C05467=1038.673,-19.331,418.240,169.034,37.910,157.122
C05468=1038.665,-19.613,418.256,169.031,37.909,157.122
C05469=1038.659,-19.895,418.271,169.029,37.909,157.121
C05470=1038.651,-20.177,418.287,169.026,37.909,157.121
C05471=1038.645,-20.426,418.300,169.024,37.909,157.121
C05472=1038.639,-20.676,418.314,169.022,37.908,157.121
C05473=1038.632,-20.925,418.328,169.019,37.908,157.121
C05474=1038.625,-21.175,418.342,169.017,37.908,157.121
C05475=1038.620,-21.425,418.356,169.014,37.907,157.121
C05476=1038.613,-21.674,418.370,169.012,37.907,157.121
C05477=1038.607,-21.923,418.384,169.010,37.907,157.121
C05478=1038.600,-22.173,418.398,169.008,37.907,157.121
C05479=1038.594,-22.423,418.411,169.006,37.906,157.121
C05480=1038.588,-22.672,418.426,169.004,37.906,157.121
C05481=1038.582,-22.922,418.439,169.001,37.906,157.120
C05482=1038.575,-23.171,418.453,168.999,37.905,157.120
C05483=1038.569,-23.421,418.467,168.997,37.905,157.120
C05484=1038.563,-23.670,418.480,168.995,37.905,157.120
C05485=1038.556,-23.920,418.494,168.993,37.905,157.120
C05486=1038.551,-24.169,418.508,168.990,37.904,157.120
C05487=1038.544,-24.419,418.522,168.988,37.904,157.120
C05488=1038.538,-24.669,418.535,168.986,37.904,157.120
C05489=1038.532,-24.918,418.549,168.984,37.904,157.120
C05490=1038.525,-25.167,418.563,168.981,37.903,157.120
C05491=1038.519,-25.417,418.577,168.978,37.903,157.120
C05492=1038.513,-25.666,418.591,168.976,37.903,157.119
C05493=1038.506,-25.916,418.604,168.974,37.902,157.119
C05494=1038.500,-26.166,418.617,168.972,37.902,157.119
C05495=1038.494,-26.416,418.632,168.970,37.902,157.119
C05496=1038.488,-26.665,418.645,168.967,37.902,157.119
C05497=1038.482,-26.915,418.659,168.965,37.901,157.119
C05498=1038.476,-27.165,418.672,168.963,37.901,157.119
C05499=1038.469,-27.414,418.686,168.961,37.901,157.119
C05500=1038.463,-27.664,418.699,168.958,37.901,157.119
C05501=1038.456,-27.913,418.713,168.956,37.900,157.119
C05502=1038.450,-28.162,418.727,168.954,37.900,157.119
C05503=1038.443,-28.412,418.740,168.952,37.900,157.119
C05504=1038.437,-28.661,418.753,168.949,37.900,157.119
C05505=1038.431,-28.911,418.766,168.947,37.900,157.119
C05506=1038.425,-29.161,418.780,168.944,37.899,157.118
C05507=1038.419,-29.410,418.794,168.942,37.899,157.118
C05508=1038.412,-29.660,418.807,168.939,37.900,157.118
C05509=1038.406,-29.910,418.820,168.937,37.899,157.118
C05510=1038.399,-30.159,418.834,168.935,37.899,157.118
C05511=1038.393,-30.409,418.847,168.933,37.899,157.118
C05512=1038.386,-30.658,418.861,168.930,37.899,157.118
C05513=1038.380,-30.907,418.874,168.928,37.899,157.118
C05514=1038.373,-31.157,418.888,168.926,37.898,157.118
C05515=1038.367,-31.407,418.901,168.924,37.898,157.118
C05516=1038.361,-31.656,418.914,168.921,37.898,157.118
C05517=1038.355,-31.905,418.927,168.919,37.898,157.118
C05518=1038.348,-32.155,418.941,168.917,37.898,157.118
C05519=1038.343,-32.405,418.954,168.915,37.897,157.118
C05520=1038.336,-32.655,418.967,168.912,37.897,157.117
C05521=1038.330,-32.905,418.981,168.910,37.897,157.117
C05522=1038.323,-33.154,418.994,168.908,37.897,157.117
C05523=1038.317,-33.403,419.008,168.906,37.897,157.117
C05524=1038.311,-33.652,419.021,168.903,37.896,157.117
C05525=1038.304,-33.902,419.034,168.901,37.896,157.117
C05526=1038.298,-34.152,419.047,168.899,37.896,157.117
C05527=1038.292,-34.401,419.060,168.895,37.896,157.117
C05528=1038.286,-34.651,419.074,168.893,37.896,157.117
C05529=1038.279,-34.901,419.087,168.891,37.895,157.117
C05530=1038.273,-35.150,419.100,168.889,37.896,157.117
C05531=1038.266,-35.432,419.115,168.886,37.896,157.117
C05532=1038.259,-35.712,419.130,168.883,37.895,157.117
C05533=1038.252,-35.993,419.145,168.881,37.895,157.117
C05534=1038.245,-36.275,419.160,168.878,37.895,157.116
C05535=1038.239,-36.524,419.173,168.876,37.895,157.116
C05536=1038.233,-36.773,419.186,168.874,37.895,157.116
C05537=1038.227,-37.023,419.199,168.872,37.894,157.116
C05538=1038.220,-37.273,419.212,168.869,37.894,157.116
C05539=1038.214,-37.523,419.226,168.867,37.894,157.116
C05540=1038.208,-37.772,419.239,168.865,37.894,157.116
C05541=1038.202,-38.022,419.252,168.862,37.894,157.116
C05542=1038.195,-38.271,419.265,168.860,37.893,157.116
C05543=1038.189,-38.520,419.278,168.858,37.893,157.116
C05544=1038.183,-38.771,419.291,168.856,37.893,157.116
C05545=1038.177,-39.020,419.304,168.853,37.893,157.116
C05546=1038.170,-39.269,419.318,168.851,37.893,157.116
C05547=1038.164,-39.519,419.330,168.849,37.893,157.116
C05548=1038.157,-39.768,419.343,168.846,37.893,157.116
C05549=1038.151,-40.019,419.356,168.843,37.893,157.116
C05550=1038.145,-40.268,419.369,168.841,37.893,157.116
C05551=1038.139,-40.518,419.382,168.838,37.893,157.116
C05552=1038.132,-40.767,419.394,168.836,37.893,157.116
C05553=1038.126,-41.016,419.407,168.834,37.893,157.116
C05554=1038.120,-41.266,419.420,168.831,37.892,157.115
C05555=1038.113,-41.516,419.434,168.829,37.892,157.115
C05556=1038.106,-41.766,419.446,168.827,37.893,157.115
C05557=1038.100,-42.015,419.459,168.824,37.893,157.115
C05558=1038.094,-42.265,419.471,168.822,37.892,157.115
C05559=1038.088,-42.514,419.485,168.820,37.892,157.115
C05560=1038.082,-42.764,419.497,168.817,37.892,157.115
C05561=1038.075,-43.013,419.510,168.815,37.892,157.115
C05562=1038.069,-43.263,419.522,168.813,37.892,157.115
C05563=1038.062,-43.513,419.536,168.810,37.892,157.115
C05564=1038.056,-43.763,419.549,168.808,37.892,157.115
C05565=1038.050,-44.012,419.561,168.805,37.892,157.115
C05566=1038.044,-44.261,419.574,168.803,37.892,157.115
C05567=1038.038,-44.511,419.586,168.801,37.892,157.115
C05568=1038.031,-44.761,419.600,168.798,37.892,157.115
C05569=1038.025,-45.010,419.612,168.796,37.892,157.115
C05570=1038.019,-45.259,419.625,168.794,37.892,157.115
C05571=1038.013,-45.509,419.638,168.791,37.892,157.115
C05572=1038.007,-45.759,419.650,168.789,37.891,157.115
C05573=1038.000,-46.008,419.663,168.787,37.891,157.114
C05574=1037.994,-46.258,419.675,168.784,37.891,157.114
C05575=1037.988,-46.508,419.688,168.782,37.892,157.114
C05576=1037.982,-46.757,419.701,168.780,37.892,157.114
C05577=1037.975,-47.007,419.713,168.777,37.891,157.114
C05578=1037.969,-47.256,419.726,168.775,37.891,157.114
C05579=1037.963,-47.506,419.739,168.773,37.891,157.114
C05580=1037.956,-47.755,419.751,168.770,37.891,157.114
C05581=1037.950,-48.005,419.764,168.768,37.891,157.114
C05582=1037.944,-48.255,419.777,168.764,37.891,157.114
C05583=1037.938,-48.504,419.789,168.762,37.891,157.114
C05584=1037.932,-48.754,419.801,168.760,37.891,157.114
C05585=1037.926,-49.003,419.814,168.757,37.891,157.114
C05586=1037.920,-49.253,419.827,168.755,37.891,157.114
C05587=1037.914,-49.503,419.840,168.753,37.891,157.114
C05588=1037.907,-49.752,419.852,168.750,37.891,157.114
C05589=1037.901,-50.002,419.865,168.748,37.891,157.114
C05590=1037.895,-50.252,419.877,168.746,37.891,157.114
C05591=1037.888,-50.501,419.889,168.743,37.891,157.114
C05592=1037.882,-50.751,419.902,168.741,37.891,157.114
C05593=1037.875,-51.000,419.915,168.738,37.891,157.114
C05594=1037.870,-51.250,419.927,168.736,37.891,157.114
C05595=1037.862,-51.532,419.940,168.733,37.891,157.114
C05596=1037.854,-51.813,419.955,168.730,37.891,157.114
C05597=1037.847,-52.095,419.968,168.728,37.892,157.114
C05598=1037.841,-52.376,419.982,168.725,37.892,157.114
C05599=1037.834,-52.626,419.994,168.722,37.892,157.114
C05600=1037.827,-52.875,420.006,168.720,37.892,157.114
C05601=1037.821,-53.125,420.019,168.718,37.892,157.114
C05602=1037.815,-53.375,420.031,168.715,37.892,157.113
C05603=1037.809,-53.624,420.043,168.713,37.892,157.113
C05604=1037.802,-53.874,420.055,168.710,37.892,157.113
C05605=1037.796,-54.124,420.067,168.708,37.892,157.113
C05606=1037.790,-54.373,420.080,168.705,37.892,157.113
C05607=1037.783,-54.623,420.092,168.703,37.893,157.114
C05608=1037.776,-54.873,420.104,168.701,37.893,157.113
C05609=1037.770,-55.122,420.116,168.698,37.893,157.113
C05610=1037.764,-55.372,420.128,168.696,37.893,157.113
C05611=1037.757,-55.622,420.140,168.693,37.893,157.113
C05612=1037.751,-55.872,420.153,168.691,37.894,157.113
C05613=1037.745,-56.121,420.165,168.688,37.894,157.113
C05614=1037.739,-56.370,420.176,168.686,37.894,157.113
C05615=1037.733,-56.620,420.189,168.683,37.894,157.113
C05616=1037.726,-56.869,420.201,168.681,37.894,157.113
C05617=1037.719,-57.119,420.213,168.679,37.894,157.113
C05618=1037.713,-57.369,420.225,168.676,37.894,157.113
C05619=1037.707,-57.618,420.237,168.674,37.894,157.113
C05620=1037.700,-57.868,420.249,168.671,37.894,157.113
C05621=1037.694,-58.118,420.262,168.669,37.895,157.113
C05622=1037.688,-58.367,420.273,168.666,37.895,157.113
C05623=1037.682,-58.617,420.285,168.664,37.895,157.113
C05624=1037.676,-58.867,420.297,168.661,37.895,157.113
C05625=1037.669,-59.116,420.309,168.659,37.895,157.113
C05626=1037.663,-59.366,420.321,168.656,37.895,157.113
C05627=1037.657,-59.616,420.334,168.654,37.896,157.113
C05628=1037.651,-59.865,420.345,168.652,37.896,157.113
C05629=1037.644,-60.114,420.357,168.649,37.896,157.113
C05630=1037.638,-60.365,420.369,168.647,37.896,157.113
C05631=1037.632,-60.614,420.381,168.644,37.896,157.113
C05632=1037.625,-60.864,420.393,168.642,37.897,157.113
C05633=1037.619,-61.113,420.405,168.639,37.897,157.113
C05634=1037.613,-61.363,420.417,168.637,37.897,157.113
C05635=1037.607,-61.613,420.428,168.634,37.897,157.113
C05636=1037.600,-61.862,420.440,168.632,37.897,157.113
C05637=1037.595,-62.112,420.453,168.629,37.897,157.113
C05638=1037.588,-62.361,420.465,168.627,37.897,157.113
C05639=1037.582,-62.611,420.476,168.624,37.897,157.113
C05640=1037.575,-62.861,420.488,168.622,37.897,157.113
C05641=1037.569,-63.111,420.500,168.619,37.897,157.113
C05642=1037.563,-63.360,420.512,168.617,37.898,157.113
C05643=1037.557,-63.609,420.524,168.614,37.898,157.113
C05644=1037.551,-63.860,420.536,168.612,37.898,157.113
C05645=1037.545,-64.109,420.547,168.610,37.898,157.113
C05646=1037.538,-64.358,420.559,168.607,37.899,157.113
C05647=1037.532,-64.608,420.570,168.605,37.899,157.113
C05648=1037.526,-64.858,420.583,168.602,37.899,157.113
C05649=1037.520,-65.107,420.595,168.600,37.899,157.113
C05650=1037.514,-65.357,420.606,168.597,37.899,157.113
C05651=1037.507,-65.607,420.618,168.595,37.900,157.113
C05652=1037.502,-65.856,420.630,168.592,37.900,157.113
C05653=1037.495,-66.106,420.641,168.590,37.900,157.113
C05654=1037.489,-66.356,420.653,168.587,37.900,157.113
C05655=1037.483,-66.605,420.665,168.585,37.900,157.113
C05656=1037.477,-66.855,420.677,168.582,37.900,157.113
C05657=1037.470,-67.105,420.689,168.580,37.900,157.113
C05658=1037.465,-67.354,420.699,168.577,37.900,157.113
C05659=1037.457,-67.637,420.714,168.574,37.901,157.113
C05660=1037.450,-67.920,420.727,168.572,37.901,157.113
C05661=1037.444,-68.202,420.740,168.569,37.901,157.113
C05662=1037.437,-68.485,420.753,168.566,37.901,157.113
C05663=1037.431,-68.735,420.765,168.564,37.901,157.113
C05664=1037.425,-68.985,420.776,168.561,37.902,157.113
C05665=1037.419,-69.234,420.788,168.559,37.902,157.113
C05666=1037.412,-69.484,420.799,168.556,37.902,157.113
C05667=1037.406,-69.733,420.811,168.554,37.902,157.113
C05668=1037.401,-69.984,420.823,168.551,37.903,157.113
C05669=1037.394,-70.233,420.835,168.549,37.903,157.113
C05670=1037.388,-70.483,420.845,168.546,37.903,157.113
C05671=1037.382,-70.732,420.857,168.544,37.903,157.113
C05672=1037.377,-70.982,420.869,168.541,37.903,157.113
C05673=1037.370,-71.232,420.881,168.539,37.904,157.113
C05674=1037.364,-71.481,420.892,168.536,37.904,157.113
C05675=1037.358,-71.731,420.904,168.534,37.904,157.113
C05676=1037.351,-71.981,420.915,168.531,37.904,157.113
C05677=1037.346,-72.231,420.926,168.529,37.904,157.113
C05678=1037.340,-72.480,420.938,168.526,37.904,157.113
C05679=1037.334,-72.730,420.949,168.524,37.905,157.113
C05680=1037.327,-72.979,420.961,168.521,37.905,157.113
C05681=1037.321,-73.229,420.972,168.519,37.905,157.113
C05682=1037.315,-73.479,420.985,168.516,37.905,157.113
C05683=1037.310,-73.728,420.996,168.514,37.905,157.113
C05684=1037.303,-73.978,421.007,168.511,37.905,157.113
C05685=1037.297,-74.227,421.018,168.508,37.906,157.113
C05686=1037.291,-74.477,421.030,168.506,37.906,157.113
C05687=1037.285,-74.727,421.040,168.503,37.906,157.113
C05688=1037.279,-74.977,421.052,168.501,37.907,157.113
C05689=1037.273,-75.226,421.063,168.498,37.907,157.113
C05690=1037.267,-75.476,421.075,168.496,37.908,157.113
C05691=1037.261,-75.726,421.085,168.493,37.908,157.113
C05692=1037.254,-75.975,421.097,168.491,37.908,157.113
C05693=1037.248,-76.225,421.108,168.488,37.909,157.113
C05694=1037.242,-76.475,421.120,168.485,37.909,157.113
C05695=1037.236,-76.724,421.130,168.483,37.909,157.113
C05696=1037.229,-76.974,421.142,168.480,37.910,157.113
C05697=1037.223,-77.223,421.153,168.478,37.910,157.113
C05698=1037.217,-77.473,421.164,168.475,37.911,157.113
C05699=1037.211,-77.723,421.175,168.473,37.911,157.113
C05700=1037.205,-77.973,421.186,168.470,37.911,157.113
C05701=1037.199,-78.222,421.198,168.468,37.911,157.113
C05702=1037.192,-78.472,421.209,168.465,37.912,157.113
C05703=1037.187,-78.722,421.220,168.462,37.912,157.113
C05704=1037.180,-78.972,421.231,168.460,37.912,157.113
C05705=1037.175,-79.221,421.242,168.457,37.913,157.113
C05706=1037.169,-79.471,421.253,168.455,37.913,157.113
C05707=1037.162,-79.721,421.263,168.452,37.913,157.113
C05708=1037.156,-79.970,421.274,168.450,37.913,157.113
C05709=1037.149,-80.220,421.286,168.448,37.914,157.113
C05710=1037.144,-80.469,421.297,168.445,37.915,157.113
C05711=1037.137,-80.719,421.308,168.443,37.915,157.113
C05712=1037.131,-80.969,421.319,168.440,37.916,157.113
C05713=1037.125,-81.219,421.330,168.437,37.916,157.113
C05714=1037.118,-81.468,421.340,168.435,37.917,157.113
C05715=1037.112,-81.718,421.351,168.432,37.917,157.113
C05716=1037.106,-81.968,421.362,168.430,37.918,157.114
C05717=1037.099,-82.217,421.373,168.427,37.918,157.114
C05718=1037.093,-82.467,421.384,168.424,37.918,157.114
C05719=1037.087,-82.716,421.395,168.422,37.919,157.114
C05720=1037.080,-82.966,421.405,168.419,37.919,157.114
C05721=1037.075,-83.216,421.416,168.417,37.920,157.114
C05722=1037.069,-83.465,421.427,168.414,37.920,157.114
C05723=1037.062,-83.751,421.439,168.411,37.921,157.114
C05724=1037.054,-84.036,421.452,168.408,37.922,157.114
C05725=1037.047,-84.321,421.464,168.405,37.922,157.114
C05726=1037.040,-84.606,421.476,168.402,37.922,157.114
C05727=1037.034,-84.855,421.486,168.399,37.923,157.114
C05728=1037.028,-85.105,421.497,168.397,37.923,157.114
C05729=1037.022,-85.355,421.508,168.394,37.924,157.114
C05730=1037.015,-85.604,421.519,168.391,37.925,157.114
C05731=1037.009,-85.854,421.529,168.389,37.925,157.114
C05732=1037.003,-86.104,421.541,168.387,37.926,157.114
C05733=1036.997,-86.354,421.550,168.385,37.926,157.114
C05734=1036.991,-86.603,421.561,168.382,37.927,157.114
C05735=1036.985,-86.853,421.572,168.379,37.927,157.114
C05736=1036.978,-87.102,421.583,168.377,37.927,157.114
C05737=1036.973,-87.352,421.594,168.374,37.928,157.114
C05738=1036.965,-87.602,421.604,168.371,37.928,157.114
C05739=1036.960,-87.852,421.614,168.369,37.929,157.115
C05740=1036.954,-88.101,421.625,168.366,37.930,157.115
C05741=1036.948,-88.351,421.636,168.364,37.930,157.115
C05742=1036.941,-88.601,421.647,168.361,37.931,157.115
C05743=1036.935,-88.850,421.657,168.358,37.931,157.115
C05744=1036.930,-89.100,421.667,168.356,37.931,157.115
C05745=1036.924,-89.350,421.678,168.353,37.932,157.115
C05746=1036.917,-89.599,421.689,168.350,37.933,157.115
C05747=1036.911,-89.849,421.700,168.348,37.933,157.115
C05748=1036.905,-90.099,421.709,168.345,37.934,157.115
C05749=1036.899,-90.348,421.720,168.342,37.934,157.115
C05750=1036.893,-90.598,421.731,168.340,37.935,157.115
C05751=1036.887,-90.848,421.741,168.337,37.935,157.115
C05752=1036.881,-91.098,421.752,168.335,37.936,157.115
C05753=1036.874,-91.347,421.762,168.332,37.936,157.115
C05754=1036.869,-91.596,421.773,168.330,37.937,157.115
C05755=1036.863,-91.847,421.783,168.328,37.937,157.115
C05756=1036.856,-92.096,421.794,168.325,37.938,157.115
C05757=1036.850,-92.346,421.805,168.322,37.939,157.115
C05758=1036.844,-92.596,421.814,168.320,37.939,157.115
C05759=1036.838,-92.845,421.825,168.317,37.940,157.116
C05760=1036.832,-93.096,421.835,168.314,37.940,157.116
C05761=1036.826,-93.345,421.846,168.312,37.940,157.116
C05762=1036.820,-93.595,421.857,168.309,37.941,157.116
C05763=1036.814,-93.844,421.866,168.306,37.942,157.116
C05764=1036.808,-94.094,421.877,168.304,37.942,157.116
C05765=1036.802,-94.344,421.887,168.301,37.943,157.116
C05766=1036.796,-94.593,421.898,168.298,37.944,157.116
C05767=1036.789,-94.843,421.908,168.296,37.944,157.116
C05768=1036.784,-95.093,421.918,168.293,37.944,157.116
C05769=1036.778,-95.343,421.929,168.291,37.945,157.116
C05770=1036.772,-95.592,421.939,168.288,37.946,157.116
C05771=1036.766,-95.842,421.950,168.285,37.946,157.116
C05772=1036.760,-96.092,421.959,168.283,37.947,157.116
C05773=1036.754,-96.341,421.970,168.281,37.948,157.116
C05774=1036.748,-96.591,421.980,168.277,37.948,157.116
C05775=1036.742,-96.841,421.991,168.276,37.948,157.116
C05776=1036.736,-97.091,422.001,168.273,37.949,157.116
C05777=1036.730,-97.341,422.011,168.270,37.949,157.116
C05778=1036.724,-97.590,422.021,168.268,37.950,157.117
C05779=1036.718,-97.840,422.032,168.265,37.951,157.117
C05780=1036.712,-98.090,422.041,168.262,37.952,157.117
C05781=1036.706,-98.339,422.051,168.260,37.952,157.117
C05782=1036.700,-98.589,422.062,168.257,37.953,157.117
C05783=1036.694,-98.839,422.071,168.254,37.954,157.117
C05784=1036.687,-99.088,422.082,168.251,37.955,157.117
C05785=1036.682,-99.338,422.092,168.249,37.955,157.117
C05786=1036.676,-99.588,422.101,168.246,37.955,157.117
C05787=1036.668,-99.874,422.113,168.243,37.956,157.117
C05788=1036.661,-100.162,422.125,168.240,37.957,157.117
C05789=1036.654,-100.449,422.136,168.238,37.958,157.117
C05790=1036.647,-100.737,422.148,168.235,37.959,157.118
C05791=1036.641,-100.987,422.158,168.232,37.959,157.118
C05792=1036.635,-101.236,422.168,168.229,37.960,157.118
C05793=1036.629,-101.486,422.178,168.226,37.961,157.118
C05794=1036.623,-101.736,422.187,168.224,37.962,157.118
C05795=1036.617,-101.986,422.197,168.221,37.962,157.118
C05796=1036.611,-102.235,422.208,168.218,37.963,157.118
C05797=1036.605,-102.485,422.217,168.216,37.964,157.118
C05798=1036.598,-102.734,422.227,168.213,37.965,157.118
C05799=1036.593,-102.984,422.238,168.210,37.965,157.118
C05800=1036.586,-103.234,422.247,168.208,37.966,157.118
C05801=1036.580,-103.484,422.257,168.205,37.967,157.118
C05802=1036.575,-103.734,422.267,168.203,37.968,157.119
C05803=1036.569,-103.983,422.277,168.200,37.969,157.119
C05804=1036.562,-104.233,422.287,168.198,37.969,157.119
C05805=1036.556,-104.482,422.296,168.195,37.970,157.119
C05806=1036.550,-104.732,422.306,168.192,37.971,157.119
C05807=1036.544,-104.982,422.316,168.190,37.972,157.119
C05808=1036.538,-105.232,422.326,168.187,37.972,157.119
C05809=1036.532,-105.482,422.335,168.184,37.972,157.119
C05810=1036.526,-105.731,422.346,168.181,37.973,157.119
C05811=1036.521,-105.981,422.355,168.179,37.974,157.119
C05812=1036.515,-106.230,422.365,168.176,37.975,157.119
C05813=1036.508,-106.480,422.375,168.173,37.976,157.119
C05814=1036.502,-106.730,422.384,168.171,37.977,157.120
C05815=1036.496,-106.980,422.394,168.169,37.978,157.120
C05816=1036.490,-107.230,422.403,168.166,37.978,157.120
C05817=1036.484,-107.480,422.413,168.163,37.979,157.120
C05818=1036.478,-107.729,422.423,168.161,37.980,157.120
C05819=1036.472,-107.979,422.433,168.158,37.981,157.120
C05820=1036.466,-108.229,422.442,168.155,37.982,157.120
C05821=1036.460,-108.479,422.452,168.152,37.982,157.120
C05822=1036.454,-108.729,422.461,168.150,37.983,157.120
C05823=1036.448,-108.978,422.470,168.147,37.984,157.120
C05824=1036.442,-109.228,422.480,168.144,37.985,157.120
C05825=1036.436,-109.477,422.490,168.141,37.985,157.121
C05826=1036.430,-109.727,422.499,168.140,37.987,157.121
C05827=1036.423,-109.977,422.509,168.137,37.988,157.121
C05828=1036.417,-110.227,422.518,168.134,37.988,157.121
C05829=1036.411,-110.477,422.528,168.131,37.989,157.121
C05830=1036.405,-110.726,422.537,168.129,37.990,157.121
C05831=1036.399,-110.975,422.547,168.126,37.991,157.121
C05832=1036.393,-111.225,422.556,168.123,37.991,157.121
C05833=1036.388,-111.475,422.566,168.120,37.993,157.121
C05834=1036.381,-111.725,422.576,168.118,37.994,157.122
C05835=1036.375,-111.975,422.585,168.115,37.994,157.122
C05836=1036.369,-112.225,422.595,168.112,37.995,157.122
C05837=1036.364,-112.474,422.604,168.110,37.996,157.122
C05838=1036.358,-112.724,422.613,168.108,37.997,157.122
C05839=1036.352,-112.974,422.623,168.105,37.997,157.122
C05840=1036.345,-113.224,422.632,168.102,37.999,157.122
C05841=1036.339,-113.474,422.642,168.099,38.000,157.122
C05842=1036.334,-113.723,422.651,168.097,38.000,157.122
C05843=1036.327,-113.973,422.661,168.094,38.001,157.122
C05844=1036.321,-114.222,422.670,168.091,38.002,157.122
C05845=1036.315,-114.473,422.679,168.088,38.003,157.123
C05846=1036.310,-114.722,422.688,168.085,38.004,157.123
C05847=1036.304,-114.972,422.698,168.084,38.005,157.123
C05848=1036.297,-115.221,422.707,168.081,38.006,157.123
C05849=1036.291,-115.472,422.716,168.078,38.007,157.123
C05850=1036.285,-115.721,422.725,168.075,38.008,157.123
C05851=1036.279,-116.007,422.736,168.072,38.009,157.123
C05852=1036.272,-116.294,422.747,168.069,38.010,157.124
C05853=1036.264,-116.580,422.757,168.066,38.011,157.124
C05854=1036.258,-116.867,422.768,168.063,38.012,157.124
C05855=1036.252,-117.117,422.777,168.060,38.013,157.124
C05856=1036.246,-117.367,422.786,168.058,38.014,157.124
C05857=1036.240,-117.616,422.795,168.055,38.015,157.124
C05858=1036.233,-117.866,422.804,168.052,38.016,157.124
C05859=1036.227,-118.116,422.813,168.050,38.017,157.124
C05860=1036.222,-118.365,422.822,168.047,38.018,157.124
C05861=1036.216,-118.615,422.832,168.044,38.019,157.125
C05862=1036.210,-118.865,422.841,168.041,38.020,157.125
C05863=1036.204,-119.114,422.850,168.039,38.021,157.125
C05864=1036.197,-119.364,422.859,168.036,38.022,157.125
C05865=1036.191,-119.614,422.868,168.034,38.023,157.125
C05866=1036.185,-119.864,422.877,168.031,38.024,157.125
C05867=1036.180,-120.114,422.886,168.028,38.025,157.125
C05868=1036.174,-120.364,422.895,168.026,38.026,157.125
C05869=1036.168,-120.613,422.905,168.023,38.027,157.126
C05870=1036.162,-120.863,422.913,168.020,38.028,157.126
C05871=1036.155,-121.113,422.922,168.017,38.029,157.126
C05872=1036.150,-121.362,422.931,168.014,38.030,157.126
C05873=1036.144,-121.612,422.940,168.012,38.031,157.126
C05874=1036.138,-121.863,422.949,168.010,38.032,157.126
C05875=1036.132,-122.111,422.958,168.007,38.033,157.126
C05876=1036.126,-122.362,422.967,168.004,38.034,157.126
C05877=1036.120,-122.612,422.976,168.001,38.036,157.127
C05878=1036.115,-122.861,422.985,167.999,38.036,157.127
C05879=1036.108,-123.111,422.994,167.996,38.037,157.127
C05880=1036.102,-123.360,423.002,167.993,38.039,157.127
C05881=1036.096,-123.610,423.012,167.990,38.039,157.127
C05882=1036.090,-123.861,423.021,167.988,38.041,157.127
C05883=1036.085,-124.110,423.030,167.986,38.042,157.127
C05884=1036.078,-124.360,423.038,167.983,38.042,157.127
C05885=1036.073,-124.610,423.047,167.980,38.044,157.128
C05886=1036.067,-124.859,423.056,167.977,38.045,157.128
C05887=1036.060,-125.109,423.064,167.974,38.046,157.128
C05888=1036.055,-125.359,423.074,167.972,38.047,157.128
C05889=1036.049,-125.609,423.082,167.969,38.048,157.128
C05890=1036.043,-125.858,423.090,167.966,38.049,157.128
C05891=1036.036,-126.108,423.100,167.964,38.050,157.129
C05892=1036.031,-126.358,423.108,167.961,38.051,157.129
C05893=1036.025,-126.608,423.117,167.958,38.053,157.129
C05894=1036.019,-126.857,423.126,167.956,38.053,157.129
C05895=1036.012,-127.107,423.134,167.953,38.055,157.129
C05896=1036.007,-127.356,423.143,167.950,38.056,157.129
C05897=1036.001,-127.607,423.152,167.947,38.057,157.129
C05898=1035.995,-127.856,423.160,167.945,38.059,157.130
C05899=1035.990,-128.106,423.170,167.943,38.059,157.130
C05900=1035.985,-128.356,423.180,167.940,38.059,157.130
C05901=1035.981,-128.605,423.190,167.938,38.059,157.129
C05902=1035.978,-128.855,423.201,167.935,38.058,157.129
C05903=1035.975,-129.105,423.213,167.933,38.057,157.129
C05904=1035.974,-129.355,423.224,167.931,38.056,157.129
C05905=1035.973,-129.605,423.238,167.929,38.054,157.128
C05906=1035.973,-129.855,423.251,167.927,38.051,157.128
C05907=1035.974,-130.105,423.265,167.925,38.048,157.127
C05908=1035.975,-130.354,423.280,167.923,38.045,157.127
C05909=1035.977,-130.604,423.294,167.922,38.041,157.126
C05910=1035.980,-130.854,423.311,167.920,38.037,157.125
C05911=1035.983,-131.105,423.327,167.920,38.032,157.125
C05912=1035.987,-131.355,423.343,167.918,38.027,157.124
C05913=1035.992,-131.605,423.361,167.917,38.021,157.123
C05914=1035.998,-131.854,423.379,167.916,38.015,157.122
C05915=1035.662,-131.880,423.102,167.867,38.229,157.157
C05916=1035.656,-131.630,423.084,167.868,38.235,157.158
C05917=1035.652,-131.380,423.066,167.870,38.241,157.159
C05918=1035.647,-131.130,423.050,167.871,38.246,157.160
C05919=1035.644,-130.879,423.032,167.872,38.251,157.160
C05920=1035.642,-130.629,423.017,167.874,38.255,157.161
C05921=1035.640,-130.379,423.002,167.876,38.258,157.162
C05922=1035.638,-130.130,422.988,167.877,38.262,157.163
C05923=1035.638,-129.880,422.974,167.879,38.265,157.163
C05924=1035.638,-129.630,422.960,167.881,38.268,157.164
C05925=1035.638,-129.379,422.948,167.882,38.270,157.164
C05926=1035.640,-129.130,422.935,167.885,38.272,157.164
C05927=1035.643,-128.880,422.924,167.887,38.272,157.164
C05928=1035.646,-128.630,422.913,167.889,38.273,157.165
C05929=1035.649,-128.380,422.902,167.892,38.273,157.165
C05930=1035.654,-128.131,422.892,167.894,38.273,157.165
C05931=1035.659,-127.881,422.883,167.897,38.272,157.165
C05932=1035.665,-127.631,422.874,167.899,38.271,157.164
C05933=1035.670,-127.382,422.866,167.902,38.270,157.164
C05934=1035.677,-127.132,422.857,167.905,38.269,157.164
C05935=1035.682,-126.883,422.848,167.907,38.268,157.164
C05936=1035.688,-126.632,422.839,167.910,38.266,157.164
C05937=1035.694,-126.383,422.831,167.913,38.266,157.164
C05938=1035.700,-126.133,422.822,167.916,38.264,157.164
C05939=1035.707,-125.883,422.814,167.918,38.263,157.163
C05940=1035.712,-125.633,422.805,167.921,38.262,157.163
C05941=1035.718,-125.383,422.796,167.924,38.260,157.163
C05942=1035.724,-125.134,422.788,167.926,38.260,157.163
C05943=1035.731,-124.884,422.778,167.929,38.258,157.163
C05944=1035.737,-124.596,422.768,167.932,38.257,157.163
C05945=1035.745,-124.306,422.758,167.935,38.256,157.163
C05946=1035.751,-124.017,422.748,167.939,38.254,157.162
C05947=1035.758,-123.728,422.738,167.942,38.253,157.162
C05948=1035.763,-123.479,422.728,167.945,38.252,157.162
C05949=1035.770,-123.229,422.720,167.946,38.251,157.162
C05950=1035.776,-122.980,422.711,167.949,38.250,157.162
C05951=1035.781,-122.729,422.702,167.952,38.248,157.162
C05952=1035.788,-122.480,422.693,167.955,38.248,157.162
C05953=1035.794,-122.230,422.685,167.958,38.247,157.161
C05954=1035.800,-121.980,422.675,167.961,38.245,157.161
C05955=1035.806,-121.730,422.666,167.963,38.245,157.161
C05956=1035.811,-121.481,422.657,167.966,38.243,157.161
C05957=1035.817,-121.230,422.648,167.968,38.242,157.161
C05958=1035.823,-120.982,422.640,167.971,38.241,157.161
C05959=1035.829,-120.731,422.631,167.974,38.240,157.161
C05960=1035.835,-120.481,422.621,167.976,38.239,157.161
C05961=1035.841,-120.232,422.613,167.979,38.238,157.160
C05962=1035.847,-119.982,422.603,167.982,38.237,157.160
C05963=1035.853,-119.732,422.594,167.985,38.236,157.160
C05964=1035.859,-119.483,422.586,167.988,38.235,157.160
C05965=1035.865,-119.233,422.576,167.991,38.234,157.160
C05966=1035.871,-118.982,422.567,167.992,38.232,157.160
C05967=1035.877,-118.733,422.558,167.995,38.232,157.160
C05968=1035.883,-118.484,422.548,167.998,38.231,157.160
C05969=1035.889,-118.233,422.540,168.001,38.229,157.159
C05970=1035.896,-117.984,422.531,168.004,38.229,157.159
C05971=1035.901,-117.735,422.521,168.006,38.228,157.159
C05972=1035.907,-117.486,422.512,168.009,38.226,157.159
C05973=1035.913,-117.237,422.504,168.012,38.226,157.159
C05974=1035.919,-116.988,422.494,168.014,38.225,157.159
C05975=1035.925,-116.740,422.485,168.017,38.223,157.159
C05976=1035.931,-116.492,422.476,168.019,38.223,157.159
C05977=1035.937,-116.243,422.467,168.022,38.222,157.159
C05978=1035.942,-115.994,422.458,168.025,38.220,157.158
C05979=1035.949,-115.746,422.448,168.028,38.220,157.158
C05980=1035.955,-115.496,422.439,168.030,38.219,157.158
C05981=1035.961,-115.246,422.430,168.033,38.217,157.158
C05982=1035.967,-114.996,422.421,168.036,38.217,157.158
C05983=1035.973,-114.747,422.411,168.038,38.216,157.158
C05984=1035.979,-114.497,422.402,168.041,38.215,157.158
C05985=1035.985,-114.246,422.393,168.043,38.214,157.158
C05986=1035.990,-113.997,422.384,168.046,38.213,157.157
C05987=1035.997,-113.748,422.374,168.049,38.212,157.157
C05988=1036.003,-113.498,422.364,168.052,38.211,157.157
C05989=1036.009,-113.248,422.355,168.055,38.210,157.157
C05990=1036.015,-112.999,422.346,168.057,38.209,157.157
C05991=1036.020,-112.748,422.337,168.060,38.208,157.157
C05992=1036.027,-112.499,422.327,168.063,38.207,157.157
C05993=1036.033,-112.249,422.318,168.065,38.207,157.157
C05994=1036.039,-111.999,422.308,168.067,38.205,157.157
C05995=1036.045,-111.750,422.299,168.070,38.204,157.156
C05996=1036.051,-111.500,422.289,168.073,38.203,157.156
C05997=1036.057,-111.250,422.280,168.076,38.203,157.156
C05998=1036.063,-111.001,422.270,168.079,38.202,157.156
C05999=1036.069,-110.751,422.261,168.081,38.200,157.156
C06000=1036.075,-110.501,422.251,168.084,38.200,157.156
C06001=1036.081,-110.251,422.243,168.087,38.199,157.156
C06002=1036.087,-110.001,422.233,168.090,38.198,157.156
C06003=1036.093,-109.752,422.224,168.091,38.197,157.156
C06004=1036.099,-109.502,422.214,168.094,38.197,157.156
C06005=1036.105,-109.252,422.204,168.097,38.195,157.155
C06006=1036.111,-109.002,422.194,168.100,38.194,157.155
C06007=1036.117,-108.752,422.185,168.102,38.194,157.155
C06008=1036.123,-108.502,422.175,168.105,38.193,157.155
C06009=1036.129,-108.253,422.166,168.108,38.192,157.155
C06010=1036.135,-108.003,422.156,168.111,38.191,157.155
C06011=1036.141,-107.754,422.147,168.114,38.190,157.155
C06012=1036.147,-107.504,422.137,168.115,38.189,157.155
C06013=1036.153,-107.254,422.128,168.118,38.188,157.155
C06014=1036.160,-107.005,422.117,168.121,38.187,157.155
C06015=1036.166,-106.755,422.108,168.124,38.187,157.154
C06016=1036.171,-106.505,422.098,168.126,38.186,157.154
C06017=1036.178,-106.255,422.088,168.129,38.185,157.154
C06018=1036.184,-106.005,422.078,168.132,38.184,157.154
C06019=1036.190,-105.756,422.069,168.134,38.183,157.154
C06020=1036.196,-105.506,422.059,168.137,38.183,157.154
C06021=1036.202,-105.256,422.049,168.140,38.182,157.154
C06022=1036.207,-105.007,422.040,168.143,38.181,157.154
C06023=1036.214,-104.757,422.030,168.145,38.180,157.154
C06024=1036.220,-104.508,422.020,168.147,38.180,157.154
C06025=1036.225,-104.257,422.010,168.150,38.179,157.154
C06026=1036.231,-104.008,422.000,168.153,38.178,157.154
C06027=1036.238,-103.758,421.991,168.155,38.177,157.153
C06028=1036.244,-103.509,421.981,168.158,38.176,157.153
C06029=1036.249,-103.259,421.970,168.161,38.176,157.153
C06030=1036.256,-103.009,421.961,168.164,38.175,157.153
C06031=1036.262,-102.759,421.951,168.166,38.174,157.153
C06032=1036.268,-102.509,421.942,168.169,38.173,157.153
C06033=1036.274,-102.260,421.931,168.172,38.173,157.153
C06034=1036.280,-102.010,421.921,168.174,38.172,157.153
C06035=1036.286,-101.760,421.912,168.177,38.171,157.153
C06036=1036.292,-101.510,421.902,168.180,38.170,157.153
C06037=1036.298,-101.261,421.891,168.182,38.169,157.153
C06038=1036.304,-101.011,421.882,168.184,38.169,157.153
C06039=1036.310,-100.761,421.872,168.187,38.168,157.152
C06040=1036.317,-100.474,421.860,168.190,38.167,157.152
C06041=1036.324,-100.187,421.848,168.193,38.166,157.152
C06042=1036.332,-99.900,421.837,168.197,38.165,157.152
C06043=1036.338,-99.612,421.825,168.200,38.165,157.152
C06044=1036.345,-99.362,421.816,168.202,38.164,157.152
C06045=1036.351,-99.113,421.805,168.205,38.163,157.152
C06046=1036.357,-98.863,421.796,168.208,38.162,157.152
C06047=1036.363,-98.613,421.786,168.211,38.162,157.152
C06048=1036.369,-98.364,421.775,168.213,38.161,157.152
C06049=1036.375,-98.114,421.766,168.215,38.160,157.152
C06050=1036.381,-97.865,421.755,168.218,38.159,157.152
C06051=1036.387,-97.615,421.745,168.220,38.158,157.151
C06052=1036.393,-97.365,421.736,168.223,38.158,157.151
C06053=1036.399,-97.116,421.725,168.226,38.157,157.151
C06054=1036.405,-96.865,421.715,168.228,38.157,157.151
C06055=1036.412,-96.616,421.704,168.231,38.156,157.151
C06056=1036.417,-96.365,421.694,168.234,38.155,157.151
C06057=1036.424,-96.116,421.684,168.236,38.154,157.151
C06058=1036.429,-95.866,421.674,168.239,38.154,157.151
C06059=1036.435,-95.617,421.663,168.242,38.154,157.151
C06060=1036.441,-95.367,421.653,168.244,38.153,157.151
C06061=1036.447,-95.118,421.643,168.247,38.152,157.151
C06062=1036.453,-94.868,421.632,168.250,38.152,157.151
C06063=1036.459,-94.618,421.622,168.252,38.151,157.151
C06064=1036.466,-94.368,421.611,168.255,38.150,157.151
C06065=1036.471,-94.118,421.601,168.257,38.150,157.151
C06066=1036.478,-93.869,421.591,168.259,38.149,157.151
C06067=1036.483,-93.619,421.580,168.262,38.149,157.151
C06068=1036.489,-93.370,421.570,168.265,38.148,157.150
C06069=1036.495,-93.120,421.559,168.267,38.148,157.150
C06070=1036.501,-92.870,421.550,168.270,38.147,157.150
C06071=1036.508,-92.620,421.539,168.273,38.146,157.150
C06072=1036.513,-92.371,421.528,168.275,38.145,157.150
C06073=1036.520,-92.121,421.518,168.278,38.145,157.150
C06074=1036.525,-91.871,421.507,168.281,38.145,157.150
C06075=1036.532,-91.622,421.497,168.283,38.144,157.150
C06076=1036.537,-91.372,421.487,168.286,38.144,157.150
C06077=1036.544,-91.122,421.476,168.289,38.143,157.150
C06078=1036.550,-90.873,421.465,168.291,38.142,157.150
C06079=1036.555,-90.623,421.455,168.294,38.141,157.150
C06080=1036.562,-90.373,421.445,168.297,38.141,157.150
C06081=1036.568,-90.123,421.434,168.299,38.140,157.150
C06082=1036.574,-89.873,421.424,168.302,38.140,157.150
C06083=1036.580,-89.624,421.413,168.305,38.140,157.150
C06084=1036.586,-89.374,421.402,168.306,38.139,157.150
C06085=1036.593,-89.125,421.392,168.309,38.138,157.150
C06086=1036.598,-88.874,421.381,168.312,38.138,157.150
C06087=1036.604,-88.625,421.371,168.314,38.137,157.150
C06088=1036.611,-88.376,421.360,168.317,38.136,157.149
C06089=1036.617,-88.126,421.349,168.320,38.136,157.149
C06090=1036.623,-87.876,421.339,168.322,38.135,157.149
C06091=1036.629,-87.626,421.329,168.325,38.135,157.149
C06092=1036.635,-87.377,421.318,168.328,38.134,157.149
C06093=1036.642,-87.127,421.307,168.330,38.134,157.149
C06094=1036.647,-86.877,421.296,168.333,38.133,157.149
C06095=1036.654,-86.628,421.286,168.336,38.132,157.149
C06096=1036.660,-86.377,421.275,168.338,38.132,157.149
C06097=1036.666,-86.128,421.264,168.341,38.131,157.149
C06098=1036.672,-85.879,421.254,168.344,38.131,157.149
C06099=1036.679,-85.629,421.243,168.346,38.131,157.149
C06100=1036.684,-85.379,421.232,168.349,38.130,157.149
C06101=1036.691,-85.130,421.222,168.351,38.129,157.149
C06102=1036.697,-84.880,421.211,168.354,38.129,157.149
C06103=1036.704,-84.631,421.200,168.356,38.128,157.149
C06104=1036.710,-84.345,421.187,168.359,38.127,157.149
C06105=1036.717,-84.060,421.175,168.362,38.127,157.149
C06106=1036.724,-83.775,421.163,168.365,38.126,157.149
C06107=1036.731,-83.490,421.151,168.368,38.126,157.148
C06108=1036.738,-83.240,421.141,168.370,38.125,157.149
C06109=1036.744,-82.991,421.130,168.373,38.125,157.148
C06110=1036.750,-82.741,421.119,168.376,38.124,157.148
C06111=1036.757,-82.492,421.108,168.378,38.124,157.148
C06112=1036.762,-82.242,421.097,168.381,38.123,157.148
C06113=1036.769,-81.992,421.086,168.384,38.122,157.148
C06114=1036.775,-81.743,421.076,168.386,38.122,157.148
C06115=1036.781,-81.493,421.065,168.389,38.121,157.148
C06116=1036.787,-81.243,421.054,168.392,38.121,157.148
C06117=1036.794,-80.994,421.043,168.394,38.121,157.148
C06118=1036.800,-80.744,421.032,168.397,38.120,157.148
C06119=1036.806,-80.494,421.021,168.399,38.120,157.148
C06120=1036.813,-80.244,421.011,168.402,38.119,157.148
C06121=1036.819,-79.995,421.000,168.405,38.118,157.148
C06122=1036.825,-79.745,420.988,168.407,38.118,157.148
C06123=1036.831,-79.495,420.978,168.409,38.117,157.148
C06124=1036.836,-79.246,420.967,168.412,38.117,157.148
C06125=1036.844,-78.996,420.955,168.415,38.117,157.148
C06126=1036.850,-78.747,420.944,168.417,38.116,157.148
C06127=1036.856,-78.497,420.933,168.419,38.116,157.148
C06128=1036.862,-78.247,420.922,168.422,38.115,157.148
C06129=1036.868,-77.997,420.911,168.424,38.115,157.148
C06130=1036.874,-77.747,420.900,168.427,38.114,157.148
C06131=1036.880,-77.498,420.888,168.430,38.114,157.148
C06132=1036.886,-77.248,420.877,168.432,38.114,157.148
C06133=1036.892,-76.998,420.866,168.435,38.114,157.148
C06134=1036.898,-76.749,420.855,168.437,38.113,157.148
C06135=1036.904,-76.499,420.844,168.440,38.113,157.148
C06136=1036.911,-76.250,420.832,168.442,38.113,157.148
C06137=1036.916,-76.000,420.822,168.445,38.112,157.147
C06138=1036.923,-75.750,420.811,168.448,38.112,157.148
C06139=1036.929,-75.501,420.800,168.450,38.111,157.147
C06140=1036.936,-75.251,420.788,168.453,38.111,157.147
C06141=1036.942,-75.001,420.777,168.455,38.111,157.147
C06142=1036.948,-74.752,420.766,168.458,38.110,157.147
C06143=1036.954,-74.502,420.754,168.460,38.110,157.147
C06144=1036.960,-74.252,420.743,168.463,38.109,157.147
C06145=1036.967,-74.002,420.732,168.466,38.109,157.147
C06146=1036.973,-73.753,420.720,168.468,38.109,157.147
C06147=1036.978,-73.503,420.708,168.471,38.109,157.147
C06148=1036.984,-73.253,420.698,168.473,38.108,157.147
C06149=1036.991,-73.004,420.686,168.476,38.108,157.147
C06150=1036.996,-72.754,420.675,168.478,38.108,157.147
C06151=1037.003,-72.505,420.663,168.481,38.108,157.147
C06152=1037.008,-72.255,420.651,168.483,38.107,157.147
C06153=1037.014,-72.005,420.640,168.486,38.107,157.147
C06154=1037.020,-71.756,420.628,168.488,38.107,157.147
C06155=1037.027,-71.506,420.617,168.491,38.107,157.147
C06156=1037.033,-71.257,420.606,168.493,38.106,157.147
C06157=1037.038,-71.006,420.594,168.496,38.106,157.147
C06158=1037.045,-70.757,420.582,168.498,38.106,157.147
C06159=1037.051,-70.507,420.571,168.501,38.105,157.147
C06160=1037.057,-70.258,420.559,168.503,38.105,157.147
C06161=1037.063,-70.008,420.548,168.506,38.105,157.147
C06162=1037.069,-69.758,420.536,168.508,38.105,157.147
C06163=1037.075,-69.509,420.525,168.511,38.104,157.147
C06164=1037.081,-69.259,420.513,168.514,38.104,157.147
C06165=1037.088,-69.009,420.501,168.516,38.104,157.147
C06166=1037.093,-68.760,420.489,168.519,38.103,157.147
C06167=1037.099,-68.510,420.478,168.521,38.103,157.147
C06168=1037.106,-68.227,420.465,168.524,38.103,157.147
C06169=1037.113,-67.945,420.451,168.527,38.103,157.147
C06170=1037.121,-67.662,420.438,168.530,38.103,157.147
C06171=1037.127,-67.379,420.425,168.532,38.102,157.147
C06172=1037.134,-67.129,420.414,168.535,38.102,157.147
C06173=1037.140,-66.880,420.402,168.537,38.102,157.147
C06174=1037.146,-66.630,420.390,168.540,38.102,157.147
C06175=1037.152,-66.380,420.378,168.542,38.102,157.147
C06176=1037.158,-66.131,420.367,168.545,38.101,157.147
C06177=1037.165,-65.881,420.355,168.547,38.101,157.147
C06178=1037.170,-65.631,420.343,168.550,38.101,157.147
C06179=1037.176,-65.382,420.331,168.552,38.101,157.147
C06180=1037.183,-65.132,420.320,168.555,38.101,157.147
C06181=1037.189,-64.882,420.308,168.557,38.101,157.148
C06182=1037.195,-64.633,420.296,168.560,38.100,157.147
C06183=1037.201,-64.383,420.284,168.562,38.100,157.147
C06184=1037.208,-64.133,420.273,168.565,38.100,157.147
C06185=1037.213,-63.884,420.261,168.567,38.099,157.148
C06186=1037.220,-63.635,420.249,168.570,38.099,157.148
C06187=1037.226,-63.384,420.237,168.572,38.099,157.148
C06188=1037.232,-63.135,420.225,168.575,38.098,157.147
C06189=1037.238,-62.886,420.213,168.577,38.098,157.147
C06190=1037.244,-62.636,420.201,168.580,38.098,157.148
C06191=1037.251,-62.386,420.190,168.582,38.098,157.148
C06192=1037.257,-62.136,420.177,168.585,38.098,157.148
C06193=1037.263,-61.887,420.166,168.587,38.098,157.148
C06194=1037.269,-61.638,420.154,168.590,38.097,157.148
C06195=1037.276,-61.387,420.143,168.592,38.097,157.148
C06196=1037.282,-61.137,420.130,168.595,38.097,157.148
C06197=1037.288,-60.888,420.118,168.597,38.097,157.148
C06198=1037.294,-60.639,420.107,168.600,38.097,157.148
C06199=1037.300,-60.389,420.094,168.602,38.097,157.148
C06200=1037.307,-60.139,420.083,168.605,38.096,157.148
C06201=1037.313,-59.889,420.071,168.607,38.096,157.148
C06202=1037.320,-59.640,420.059,168.610,38.096,157.148
C06203=1037.325,-59.391,420.047,168.612,38.096,157.148
C06204=1037.332,-59.141,420.035,168.615,38.096,157.148
C06205=1037.338,-58.891,420.023,168.617,38.095,157.148
C06206=1037.344,-58.642,420.010,168.620,38.095,157.148
C06207=1037.351,-58.392,419.998,168.622,38.095,157.148
C06208=1037.357,-58.142,419.987,168.625,38.094,157.148
C06209=1037.363,-57.893,419.975,168.627,38.094,157.148
C06210=1037.369,-57.643,419.963,168.629,38.094,157.148
C06211=1037.376,-57.393,419.951,168.632,38.094,157.148
C06212=1037.382,-57.144,419.938,168.634,38.094,157.148
C06213=1037.389,-56.894,419.926,168.637,38.094,157.148
C06214=1037.395,-56.644,419.914,168.639,38.093,157.148
C06215=1037.401,-56.395,419.902,168.642,38.093,157.148
C06216=1037.408,-56.145,419.890,168.644,38.093,157.148
C06217=1037.414,-55.896,419.878,168.647,38.093,157.148
C06218=1037.420,-55.646,419.866,168.649,38.093,157.148
C06219=1037.426,-55.397,419.854,168.652,38.093,157.148
C06220=1037.433,-55.147,419.842,168.654,38.093,157.148
C06221=1037.439,-54.897,419.829,168.657,38.092,157.148
C06222=1037.446,-54.648,419.817,168.659,38.092,157.148
C06223=1037.452,-54.398,419.805,168.662,38.092,157.148
C06224=1037.458,-54.148,419.793,168.664,38.092,157.148
C06225=1037.465,-53.899,419.781,168.666,38.091,157.148
C06226=1037.471,-53.649,419.769,168.669,38.091,157.148
C06227=1037.477,-53.399,419.756,168.671,38.091,157.148
C06228=1037.484,-53.150,419.744,168.674,38.091,157.148
C06229=1037.490,-52.900,419.732,168.676,38.091,157.148
C06230=1037.496,-52.650,419.720,168.679,38.090,157.148
C06231=1037.503,-52.401,419.708,168.681,38.090,157.148
C06232=1037.510,-52.120,419.694,168.684,38.090,157.148
C06233=1037.517,-51.838,419.680,168.687,38.090,157.148
C06234=1037.524,-51.556,419.666,168.689,38.090,157.148
C06235=1037.532,-51.275,419.653,168.692,38.090,157.148
C06236=1037.538,-51.025,419.640,168.695,38.090,157.148
C06237=1037.545,-50.775,419.628,168.697,38.089,157.148
C06238=1037.552,-50.526,419.615,168.700,38.089,157.148
C06239=1037.557,-50.276,419.603,168.702,38.089,157.148
C06240=1037.563,-50.026,419.590,168.704,38.089,157.148
C06241=1037.569,-49.777,419.578,168.707,38.089,157.148
C06242=1037.576,-49.527,419.566,168.709,38.089,157.148
C06243=1037.582,-49.278,419.552,168.711,38.089,157.148
C06244=1037.587,-49.029,419.540,168.714,38.089,157.148
C06245=1037.594,-48.779,419.528,168.716,38.089,157.148
C06246=1037.600,-48.530,419.515,168.719,38.089,157.148
C06247=1037.606,-48.280,419.503,168.721,38.089,157.148
C06248=1037.612,-48.030,419.490,168.723,38.089,157.148
C06249=1037.619,-47.781,419.477,168.726,38.089,157.148
C06250=1037.625,-47.531,419.465,168.728,38.089,157.149
C06251=1037.631,-47.281,419.452,168.731,38.089,157.149
C06252=1037.637,-47.031,419.440,168.733,38.089,157.149
C06253=1037.644,-46.782,419.427,168.735,38.089,157.149
C06254=1037.650,-46.532,419.414,168.738,38.089,157.149
C06255=1037.657,-46.283,419.401,168.740,38.089,157.149
C06256=1037.663,-46.033,419.389,168.742,38.089,157.149
C06257=1037.669,-45.783,419.376,168.745,38.089,157.149
C06258=1037.675,-45.534,419.363,168.747,38.089,157.149
C06259=1037.681,-45.284,419.350,168.750,38.089,157.149
C06260=1037.688,-45.034,419.338,168.752,38.089,157.149
C06261=1037.694,-44.785,419.325,168.754,38.089,157.149
C06262=1037.700,-44.535,419.313,168.757,38.089,157.149
C06263=1037.706,-44.286,419.299,168.759,38.089,157.149
C06264=1037.713,-44.036,419.287,168.761,38.089,157.149
C06265=1037.719,-43.787,419.274,168.764,38.089,157.149
C06266=1037.725,-43.537,419.262,168.766,38.089,157.149
C06267=1037.731,-43.288,419.248,168.768,38.089,157.149
C06268=1037.737,-43.038,419.236,168.772,38.089,157.149
C06269=1037.744,-42.788,419.223,168.774,38.089,157.149
C06270=1037.751,-42.539,419.210,168.777,38.089,157.149
C06271=1037.756,-42.289,419.198,168.779,38.089,157.149
C06272=1037.763,-42.039,419.184,168.781,38.089,157.149
C06273=1037.769,-41.790,419.172,168.784,38.089,157.149
C06274=1037.776,-41.541,419.159,168.786,38.088,157.149
C06275=1037.782,-41.291,419.146,168.788,38.089,157.150
C06276=1037.788,-41.041,419.133,168.791,38.089,157.150
C06277=1037.795,-40.792,419.120,168.793,38.089,157.150
C06278=1037.801,-40.542,419.108,168.795,38.089,157.150
C06279=1037.807,-40.293,419.094,168.798,38.089,157.150
C06280=1037.813,-40.043,419.082,168.800,38.089,157.150
C06281=1037.819,-39.793,419.069,168.802,38.089,157.150
C06282=1037.827,-39.543,419.056,168.805,38.089,157.150
C06283=1037.833,-39.294,419.043,168.807,38.089,157.150
C06284=1037.839,-39.045,419.030,168.809,38.089,157.150
C06285=1037.845,-38.795,419.017,168.812,38.089,157.150
C06286=1037.851,-38.546,419.004,168.814,38.089,157.150
C06287=1037.857,-38.296,418.991,168.816,38.089,157.150
C06288=1037.864,-38.046,418.978,168.819,38.089,157.150
C06289=1037.870,-37.796,418.964,168.821,38.089,157.150
C06290=1037.876,-37.547,418.951,168.823,38.090,157.150
C06291=1037.882,-37.297,418.939,168.826,38.089,157.150
C06292=1037.889,-37.048,418.925,168.828,38.089,157.150
C06293=1037.895,-36.798,418.912,168.830,38.090,157.151
C06294=1037.901,-36.548,418.899,168.832,38.090,157.151
C06295=1037.907,-36.299,418.886,168.835,38.090,157.151
C06296=1037.915,-36.018,418.871,168.838,38.090,157.151
C06297=1037.921,-35.737,418.856,168.841,38.090,157.151
C06298=1037.928,-35.456,418.842,168.844,38.090,157.151
C06299=1037.935,-35.175,418.826,168.846,38.091,157.151
C06300=1037.942,-34.925,418.813,168.848,38.090,157.151
C06301=1037.948,-34.675,418.800,168.851,38.090,157.151
C06302=1037.954,-34.425,418.786,168.853,38.091,157.151
C06303=1037.961,-34.176,418.773,168.855,38.091,157.151
C06304=1037.967,-33.927,418.760,168.858,38.091,157.151
C06305=1037.973,-33.678,418.747,168.860,38.091,157.151
C06306=1037.980,-33.428,418.733,168.862,38.091,157.151
C06307=1037.986,-33.178,418.720,168.864,38.091,157.151
C06308=1037.992,-32.929,418.707,168.867,38.092,157.151
C06309=1037.998,-32.679,418.694,168.869,38.092,157.151
C06310=1038.005,-32.429,418.680,168.871,38.091,157.152
C06311=1038.011,-32.180,418.667,168.874,38.092,157.152
C06312=1038.017,-31.931,418.654,168.876,38.092,157.152
C06313=1038.024,-31.681,418.640,168.878,38.092,157.152
C06314=1038.030,-31.431,418.628,168.880,38.092,157.152
C06315=1038.036,-31.181,418.614,168.883,38.092,157.152
C06316=1038.042,-30.932,418.600,168.885,38.092,157.152
C06317=1038.049,-30.682,418.587,168.887,38.093,157.152
C06318=1038.055,-30.433,418.574,168.891,38.093,157.152
C06319=1038.061,-30.184,418.560,168.893,38.093,157.152
C06320=1038.068,-29.934,418.547,168.895,38.093,157.152
C06321=1038.074,-29.684,418.533,168.897,38.093,157.152
C06322=1038.080,-29.435,418.520,168.900,38.093,157.152
C06323=1038.087,-29.185,418.506,168.902,38.093,157.152
C06324=1038.093,-28.936,418.493,168.904,38.093,157.152
C06325=1038.100,-28.686,418.480,168.906,38.093,157.152
C06326=1038.106,-28.437,418.466,168.909,38.093,157.152
C06327=1038.113,-28.187,418.453,168.911,38.094,157.153
C06328=1038.119,-27.937,418.439,168.913,38.094,157.153
C06329=1038.125,-27.688,418.425,168.915,38.094,157.153
C06330=1038.131,-27.439,418.412,168.918,38.094,157.153
C06331=1038.138,-27.189,418.399,168.920,38.094,157.153
C06332=1038.144,-26.939,418.385,168.922,38.095,157.153
C06333=1038.151,-26.689,418.372,168.924,38.095,157.153
C06334=1038.156,-26.440,418.358,168.927,38.094,157.153
C06335=1038.163,-26.191,418.345,168.929,38.095,157.153
C06336=1038.169,-25.941,418.331,168.931,38.095,157.153
C06337=1038.175,-25.691,418.317,168.933,38.095,157.153
C06338=1038.182,-25.442,418.303,168.936,38.095,157.153
C06339=1038.188,-25.192,418.289,168.939,38.096,157.153
C06340=1038.194,-24.943,418.276,168.941,38.096,157.154
C06341=1038.201,-24.693,418.262,168.943,38.096,157.154
C06342=1038.207,-24.444,418.249,168.945,38.096,157.154
C06343=1038.213,-24.193,418.234,168.948,38.097,157.154
C06344=1038.219,-23.945,418.220,168.950,38.097,157.154
C06345=1038.225,-23.695,418.207,168.952,38.097,157.154
C06346=1038.232,-23.445,418.193,168.954,38.097,157.154
C06347=1038.238,-23.196,418.180,168.957,38.098,157.154
C06348=1038.244,-22.946,418.165,168.959,38.098,157.154
C06349=1038.250,-22.697,418.151,168.961,38.098,157.154
C06350=1038.257,-22.448,418.138,168.963,38.098,157.154
C06351=1038.263,-22.197,418.124,168.965,38.099,157.154
C06352=1038.269,-21.948,418.111,168.968,38.099,157.155
C06353=1038.276,-21.699,418.096,168.970,38.099,157.155
C06354=1038.282,-21.449,418.082,168.972,38.099,157.155
C06355=1038.288,-21.199,418.069,168.975,38.100,157.155
C06356=1038.295,-20.950,418.056,168.977,38.100,157.155
C06357=1038.301,-20.700,418.041,168.980,38.100,157.155
C06358=1038.307,-20.451,418.027,168.982,38.100,157.155
C06359=1038.313,-20.201,418.013,168.984,38.101,157.155
C06360=1038.320,-19.920,417.997,168.986,38.100,157.155
C06361=1038.327,-19.637,417.982,168.989,38.101,157.155
C06362=1038.335,-19.355,417.966,168.991,38.101,157.155
C06363=1038.342,-19.074,417.950,168.994,38.101,157.155
C06364=1038.349,-18.824,417.937,168.996,38.101,157.156
C06365=1038.354,-18.575,417.923,168.998,38.102,157.156
C06366=1038.361,-18.325,417.908,169.000,38.102,157.156
C06367=1038.367,-18.076,417.895,169.003,38.102,157.156
C06368=1038.374,-17.826,417.880,169.005,38.102,157.156
C06369=1038.381,-17.577,417.866,169.007,38.103,157.156
C06370=1038.386,-17.327,417.853,169.009,38.103,157.156
C06371=1038.393,-17.078,417.838,169.012,38.103,157.156
C06372=1038.399,-16.828,417.825,169.015,38.103,157.156
C06373=1038.406,-16.579,417.810,169.017,38.104,157.156
C06374=1038.412,-16.329,417.797,169.019,38.104,157.156
C06375=1038.418,-16.079,417.783,169.021,38.104,157.156
C06376=1038.425,-15.830,417.768,169.023,38.104,157.156
C06377=1038.431,-15.581,417.755,169.026,38.105,157.157
C06378=1038.438,-15.331,417.740,169.028,38.105,157.157
C06379=1038.444,-15.082,417.727,169.030,38.105,157.157
C06380=1038.450,-14.832,417.712,169.032,38.105,157.157
C06381=1038.456,-14.582,417.698,169.034,38.106,157.157
C06382=1038.463,-14.333,417.684,169.036,38.106,157.157
C06383=1038.469,-14.083,417.669,169.038,38.106,157.157
C06384=1038.475,-13.834,417.655,169.041,38.107,157.157
C06385=1038.482,-13.584,417.641,169.043,38.107,157.157
C06386=1038.488,-13.335,417.626,169.046,38.107,157.157
C06387=1038.494,-13.085,417.612,169.048,38.108,157.158
C06388=1038.500,-12.836,417.598,169.050,38.108,157.158
C06389=1038.506,-12.586,417.583,169.052,38.108,157.158
C06390=1038.513,-12.336,417.570,169.054,38.109,157.158
C06391=1038.519,-12.087,417.555,169.057,38.109,157.158
C06392=1038.525,-11.838,417.540,169.059,38.109,157.158
C06393=1038.532,-11.588,417.527,169.061,38.109,157.158
C06394=1038.538,-11.339,417.512,169.063,38.110,157.158
C06395=1038.544,-11.089,417.497,169.065,38.110,157.158
C06396=1038.551,-10.840,417.484,169.067,38.110,157.158
C06397=1038.557,-10.590,417.469,169.069,38.111,157.159
C06398=1038.563,-10.341,417.454,169.071,38.111,157.159
C06399=1038.570,-10.091,417.441,169.074,38.111,157.159
C06400=1038.576,-9.842,417.426,169.077,38.112,157.159
C06401=1038.582,-9.592,417.411,169.079,38.112,157.159
C06402=1038.589,-9.343,417.397,169.081,38.112,157.159
C06403=1038.595,-9.093,417.382,169.083,38.113,157.159
C06404=1038.601,-8.843,417.368,169.085,38.113,157.159
C06405=1038.608,-8.594,417.354,169.087,38.113,157.159
C06406=1038.614,-8.344,417.339,169.089,38.114,157.159
C06407=1038.620,-8.095,417.324,169.092,38.114,157.159
C06408=1038.626,-7.846,417.310,169.094,38.114,157.160
C06409=1038.633,-7.596,417.296,169.096,38.114,157.160
C06410=1038.639,-7.346,417.281,169.098,38.115,157.160
C06411=1038.645,-7.097,417.267,169.100,38.115,157.160
C06412=1038.652,-6.848,417.252,169.102,38.115,157.160
C06413=1038.658,-6.598,417.238,169.105,38.116,157.160
C06414=1038.665,-6.348,417.223,169.107,38.116,157.160
C06415=1038.671,-6.099,417.209,169.110,38.116,157.160
C06416=1038.678,-5.850,417.194,169.112,38.117,157.160
C06417=1038.684,-5.600,417.179,169.114,38.117,157.160
C06418=1038.691,-5.350,417.166,169.116,38.117,157.161
C06419=1038.697,-5.101,417.151,169.118,38.118,157.161
C06420=1038.703,-4.851,417.136,169.120,38.118,157.161
C06421=1038.709,-4.602,417.121,169.122,38.118,157.161
C06422=1038.716,-4.352,417.107,169.124,38.118,157.161
C06423=1038.722,-4.104,417.092,169.126,38.119,157.161
C06424=1038.730,-3.819,417.075,169.129,38.119,157.161
C06425=1038.737,-3.536,417.059,169.131,38.119,157.161
C06426=1038.744,-3.253,417.042,169.135,38.120,157.161
C06427=1038.751,-2.969,417.025,169.137,38.120,157.161
C06428=1038.757,-2.720,417.010,169.139,38.121,157.162
C06429=1038.764,-2.470,416.995,169.141,38.121,157.162
C06430=1038.769,-2.221,416.981,169.143,38.122,157.162
C06431=1038.776,-1.971,416.966,169.145,38.122,157.162
C06432=1038.782,-1.722,416.951,169.147,38.122,157.162
C06433=1038.788,-1.473,416.936,169.149,38.123,157.162
C06434=1038.794,-1.223,416.921,169.151,38.124,157.162
C06435=1038.801,-0.973,416.906,169.153,38.124,157.162
C06436=1038.807,-0.724,416.891,169.156,38.125,157.163
C06437=1038.813,-0.474,416.876,169.158,38.125,157.163
C06438=1038.819,-0.225,416.862,169.160,38.125,157.163
C06439=1038.826,0.025,416.847,169.163,38.126,157.163
C06440=1038.832,0.274,416.832,169.165,38.126,157.163
C06441=1038.838,0.524,416.817,169.167,38.127,157.163
C06442=1038.844,0.773,416.802,169.169,38.127,157.163
C06443=1038.850,1.022,416.787,169.171,38.127,157.163
C06444=1038.857,1.272,416.772,169.173,38.128,157.163
C06445=1038.864,1.521,416.757,169.175,38.128,157.164
C06446=1038.870,1.771,416.742,169.177,38.129,157.164
C06447=1038.876,2.020,416.727,169.179,38.129,157.164
C06448=1038.882,2.269,416.712,169.182,38.129,157.164
C06449=1038.888,2.519,416.697,169.184,38.130,157.164
C06450=1038.895,2.769,416.682,169.186,38.131,157.164
C06451=1038.901,3.018,416.668,169.188,38.130,157.164
C06452=1038.907,3.268,416.652,169.190,38.131,157.164
C06453=1038.914,3.517,416.636,169.192,38.132,157.165
C06454=1038.919,3.766,416.622,169.194,38.132,157.165
C06455=1038.926,4.016,416.607,169.196,38.133,157.165
C06456=1038.932,4.266,416.592,169.198,38.133,157.165
C06457=1038.939,4.515,416.577,169.200,38.133,157.165
C06458=1038.945,4.764,416.561,169.202,38.134,157.165
C06459=1038.952,5.014,416.546,169.205,38.134,157.165
C06460=1038.958,5.264,416.531,169.207,38.135,157.165
C06461=1038.964,5.513,416.516,169.209,38.135,157.165
C06462=1038.970,5.762,416.502,169.211,38.135,157.166
C06463=1038.977,6.011,416.486,169.213,38.136,157.166
C06464=1038.983,6.261,416.471,169.215,38.136,157.166
C06465=1038.990,6.511,416.456,169.218,38.136,157.166
C06466=1038.996,6.760,416.441,169.220,38.137,157.166
C06467=1039.002,7.010,416.425,169.222,38.137,157.166
C06468=1039.008,7.259,416.410,169.224,38.138,157.166
C06469=1039.015,7.509,416.395,169.227,38.139,157.166
C06470=1039.021,7.758,416.379,169.229,38.138,157.166
C06471=1039.028,8.008,416.365,169.231,38.139,157.167
C06472=1039.034,8.257,416.350,169.233,38.140,157.167
C06473=1039.041,8.507,416.335,169.235,38.140,157.167
C06474=1039.047,8.756,416.319,169.237,38.140,157.167
C06475=1039.054,9.006,416.304,169.239,38.141,157.167
C06476=1039.060,9.255,416.289,169.241,38.141,157.167
C06477=1039.066,9.504,416.274,169.243,38.142,157.167
C06478=1039.072,9.754,416.258,169.245,38.142,157.167
C06479=1039.078,10.003,416.243,169.247,38.142,157.167
C06480=1039.085,10.252,416.228,169.249,38.143,157.168
C06481=1039.091,10.502,416.213,169.252,38.143,157.168
C06482=1039.098,10.751,416.197,169.254,38.144,157.168
C06483=1039.104,11.001,416.182,169.256,38.144,157.168
C06484=1039.111,11.250,416.167,169.258,38.144,157.168
C06485=1039.117,11.499,416.151,169.260,38.145,157.168
C06486=1039.124,11.749,416.137,169.262,38.145,157.168
C06487=1039.130,11.998,416.120,169.264,38.145,157.168
C06488=1039.137,12.284,416.103,169.266,38.146,157.168
C06489=1039.144,12.569,416.086,169.269,38.146,157.169
C06490=1039.152,12.855,416.068,169.271,38.147,157.169
C06491=1039.159,13.140,416.050,169.274,38.148,157.169
C06492=1039.166,13.390,416.035,169.276,38.147,157.169
C06493=1039.173,13.639,416.020,169.278,38.148,157.169
C06494=1039.180,13.889,416.004,169.280,38.149,157.169
C06495=1039.185,14.138,415.988,169.282,38.149,157.169
C06496=1039.192,14.388,415.973,169.284,38.150,157.170
C06497=1039.199,14.637,415.957,169.286,38.150,157.170
C06498=1039.204,14.887,415.942,169.288,38.150,157.170
C06499=1039.211,15.136,415.926,169.290,38.151,157.170
C06500=1039.217,15.386,415.911,169.292,38.151,157.170
C06501=1039.223,15.635,415.895,169.294,38.152,157.170
C06502=1039.230,15.884,415.879,169.297,38.152,157.170
C06503=1039.236,16.134,415.864,169.299,38.153,157.170
C06504=1039.242,16.383,415.848,169.301,38.153,157.171
C06505=1039.249,16.633,415.833,169.303,38.154,157.171
C06506=1039.255,16.882,415.817,169.305,38.155,157.171
C06507=1039.261,17.131,415.801,169.307,38.155,157.171
C06508=1039.268,17.381,415.786,169.309,38.155,157.171
C06509=1039.274,17.630,415.770,169.311,38.156,157.171
C06510=1039.280,17.879,415.755,169.313,38.156,157.171
C06511=1039.287,18.129,415.740,169.315,38.157,157.171
C06512=1039.293,18.378,415.723,169.318,38.157,157.172
C06513=1039.300,18.628,415.707,169.320,38.158,157.172
C06514=1039.306,18.878,415.692,169.322,38.158,157.172
C06515=1039.312,19.127,415.676,169.324,38.159,157.172
C06516=1039.319,19.376,415.660,169.326,38.159,157.172
C06517=1039.325,19.626,415.645,169.328,38.159,157.172
C06518=1039.331,19.875,415.629,169.330,38.160,157.172
C06519=1039.337,20.124,415.613,169.332,38.161,157.172
C06520=1039.344,20.373,415.597,169.334,38.161,157.173
C06521=1039.350,20.623,415.582,169.335,38.162,157.173
C06522=1039.356,20.872,415.566,169.338,38.162,157.173
C06523=1039.363,21.122,415.549,169.340,38.163,157.173
C06524=1039.370,21.371,415.534,169.342,38.163,157.173
C06525=1039.375,21.621,415.518,169.344,38.164,157.173
C06526=1039.382,21.870,415.503,169.346,38.164,157.173
C06527=1039.388,22.120,415.486,169.348,38.165,157.174
C06528=1039.394,22.369,415.471,169.350,38.166,157.174
C06529=1039.400,22.618,415.454,169.352,38.166,157.174
C06530=1039.407,22.869,415.439,169.354,38.167,157.174
C06531=1039.413,23.118,415.423,169.357,38.167,157.174
C06532=1039.419,23.367,415.407,169.359,38.167,157.174
C06533=1039.426,23.616,415.391,169.361,38.168,157.174
C06534=1039.432,23.866,415.375,169.363,38.168,157.174
C06535=1039.439,24.115,415.359,169.365,38.169,157.175
C06536=1039.445,24.364,415.343,169.367,38.169,157.175
C06537=1039.452,24.614,415.327,169.369,38.170,157.175
C06538=1039.458,24.864,415.311,169.370,38.171,157.175
C06539=1039.464,25.113,415.296,169.372,38.171,157.175
C06540=1039.470,25.362,415.279,169.375,38.172,157.175
C06541=1039.476,25.611,415.263,169.377,38.172,157.175
C06542=1039.483,25.861,415.247,169.379,38.173,157.176
C06543=1039.489,26.110,415.231,169.381,38.173,157.176
C06544=1039.496,26.360,415.215,169.383,38.174,157.176
C06545=1039.502,26.609,415.199,169.385,38.174,157.176
C06546=1039.509,26.858,415.183,169.387,38.174,157.176
C06547=1039.515,27.108,415.167,169.389,38.175,157.176
C06548=1039.521,27.357,415.150,169.391,38.175,157.176
C06549=1039.528,27.606,415.135,169.393,38.176,157.176
C06550=1039.534,27.856,415.118,169.396,38.177,157.177
C06551=1039.540,28.106,415.102,169.398,38.177,157.177
C06552=1039.547,28.393,415.084,169.400,38.178,157.177
C06553=1039.555,28.679,415.065,169.402,38.178,157.177
C06554=1039.562,28.965,415.047,169.404,38.179,157.177
C06555=1039.569,29.252,415.028,169.406,38.180,157.177
C06556=1039.576,29.502,415.012,169.408,38.181,157.178
C06557=1039.582,29.751,414.996,169.410,38.181,157.178
C06558=1039.588,30.000,414.979,169.413,38.182,157.178
C06559=1039.594,30.249,414.962,169.415,38.182,157.178
C06560=1039.601,30.499,414.946,169.417,38.183,157.178
C06561=1039.607,30.749,414.930,169.419,38.183,157.178
C06562=1039.613,30.998,414.914,169.421,38.184,157.178
C06563=1039.619,31.247,414.898,169.423,38.184,157.179
C06564=1039.626,31.497,414.881,169.424,38.185,157.179
C06565=1039.632,31.746,414.865,169.426,38.186,157.179
C06566=1039.638,31.996,414.849,169.428,38.186,157.179
C06567=1039.645,32.244,414.832,169.431,38.187,157.179
C06568=1039.651,32.494,414.816,169.433,38.187,157.179
C06569=1039.657,32.744,414.799,169.435,38.188,157.179
C06570=1039.664,32.993,414.784,169.437,38.188,157.179
C06571=1039.670,33.243,414.767,169.439,38.189,157.180
C06572=1039.677,33.492,414.750,169.441,38.189,157.180
C06573=1039.683,33.741,414.734,169.443,38.190,157.180
C06574=1039.689,33.991,414.717,169.444,38.191,157.180
C06575=1039.696,34.240,414.702,169.446,38.191,157.180
C06576=1039.702,34.489,414.685,169.449,38.192,157.180
C06577=1039.709,34.739,414.668,169.451,38.192,157.180
C06578=1039.715,34.988,414.652,169.453,38.193,157.181
C06579=1039.721,35.238,414.635,169.455,38.193,157.181
C06580=1039.728,35.487,414.619,169.457,38.194,157.181
C06581=1039.734,35.736,414.602,169.459,38.194,157.181
C06582=1039.740,35.985,414.586,169.461,38.195,157.181
C06583=1039.747,36.235,414.570,169.463,38.196,157.181
C06584=1039.753,36.485,414.553,169.465,38.196,157.181
C06585=1039.760,36.733,414.537,169.467,38.197,157.182
C06586=1039.766,36.983,414.520,169.469,38.197,157.182
C06587=1039.772,37.233,414.504,169.471,38.198,157.182
C06588=1039.778,37.481,414.487,169.473,38.198,157.182
C06589=1039.785,37.731,414.470,169.475,38.199,157.182
C06590=1039.791,37.981,414.454,169.477,38.199,157.182
C06591=1039.797,38.229,414.437,169.479,38.200,157.182
C06592=1039.804,38.479,414.421,169.482,38.201,157.183
C06593=1039.810,38.729,414.404,169.483,38.202,157.183
C06594=1039.816,38.978,414.387,169.485,38.202,157.183
C06595=1039.822,39.228,414.371,169.487,38.203,157.183
C06596=1039.829,39.476,414.354,169.489,38.203,157.183
C06597=1039.835,39.726,414.337,169.491,38.204,157.183
C06598=1039.841,39.976,414.321,169.493,38.205,157.184
C06599=1039.847,40.224,414.304,169.495,38.205,157.184
C06600=1039.854,40.474,414.287,169.496,38.206,157.184
C06601=1039.860,40.723,414.270,169.499,38.206,157.184
C06602=1039.867,40.973,414.254,169.501,38.207,157.184
C06603=1039.872,41.222,414.236,169.503,38.208,157.184
C06604=1039.878,41.472,414.220,169.505,38.209,157.185
C06605=1039.885,41.721,414.203,169.507,38.209,157.185
C06606=1039.891,41.970,414.186,169.509,38.210,157.185
C06607=1039.898,42.220,414.169,169.511,38.210,157.185
C06608=1039.904,42.469,414.153,169.512,38.211,157.185
C06609=1039.910,42.718,414.136,169.515,38.211,157.185
C06610=1039.917,42.968,414.119,169.517,38.212,157.185
C06611=1039.923,43.217,414.102,169.519,38.212,157.186
C06612=1039.929,43.467,414.085,169.521,38.213,157.186
C06613=1039.935,43.716,414.068,169.523,38.214,157.186
C06614=1039.942,43.966,414.051,169.525,38.215,157.186
C06615=1039.948,44.215,414.034,169.526,38.215,157.186
C06616=1039.954,44.501,414.015,169.528,38.216,157.186
C06617=1039.962,44.788,413.995,169.532,38.217,157.187
C06618=1039.969,45.074,413.976,169.534,38.218,157.187
C06619=1039.976,45.362,413.956,169.536,38.219,157.187
C06620=1039.982,45.610,413.939,169.538,38.219,157.187
C06621=1039.988,45.859,413.922,169.539,38.220,157.187
C06622=1039.994,46.109,413.905,169.541,38.220,157.187
C06623=1040.001,46.358,413.888,169.543,38.221,157.188
C06624=1040.007,46.608,413.870,169.546,38.222,157.188
C06625=1040.013,46.857,413.854,169.548,38.223,157.188
C06626=1040.019,47.107,413.836,169.550,38.223,157.188
C06627=1040.026,47.355,413.819,169.551,38.224,157.188
C06628=1040.032,47.605,413.803,169.553,38.224,157.188
C06629=1040.038,47.854,413.785,169.555,38.226,157.189
C06630=1040.044,48.103,413.768,169.557,38.226,157.189
C06631=1040.051,48.353,413.751,169.560,38.227,157.189
C06632=1040.056,48.602,413.734,169.562,38.227,157.189
C06633=1040.063,48.852,413.717,169.563,38.228,157.189
C06634=1040.069,49.100,413.700,169.565,38.229,157.190
C06635=1040.075,49.350,413.682,169.567,38.230,157.190
C06636=1040.081,49.600,413.665,169.569,38.230,157.190
C06637=1040.088,49.849,413.648,169.571,38.231,157.190
C06638=1040.094,50.098,413.631,169.574,38.231,157.190
C06639=1040.101,50.347,413.613,169.575,38.232,157.190
C06640=1040.106,50.597,413.597,169.577,38.233,157.190
C06641=1040.113,50.847,413.579,169.579,38.234,157.191
C06642=1040.119,51.095,413.562,169.581,38.234,157.191
C06643=1040.126,51.345,413.545,169.583,38.235,157.191
C06644=1040.132,51.594,413.527,169.585,38.235,157.191
C06645=1040.138,51.843,413.510,169.586,38.236,157.191
C06646=1040.145,52.093,413.493,169.589,38.237,157.191
C06647=1040.150,52.342,413.476,169.591,38.238,157.192
C06648=1040.157,52.592,413.458,169.593,38.238,157.192
C06649=1040.163,52.841,413.441,169.595,38.239,157.192
C06650=1040.169,53.090,413.423,169.597,38.239,157.192
C06651=1040.176,53.339,413.406,169.598,38.240,157.192
C06652=1040.182,53.589,413.388,169.600,38.241,157.192
C06653=1040.188,53.839,413.372,169.603,38.241,157.193
C06654=1040.195,54.087,413.355,169.605,38.242,157.193
C06655=1040.201,54.337,413.337,169.607,38.243,157.193
C06656=1040.207,54.586,413.320,169.609,38.243,157.193
C06657=1040.214,54.835,413.303,169.610,38.244,157.193
C06658=1040.220,55.085,413.285,169.612,38.244,157.193
C06659=1040.226,55.334,413.268,169.614,38.245,157.193
C06660=1040.233,55.583,413.250,169.616,38.246,157.194
C06661=1040.239,55.832,413.233,169.619,38.247,157.194
C06662=1040.245,56.082,413.215,169.621,38.247,157.194
C06663=1040.252,56.331,413.198,169.622,38.248,157.194
C06664=1040.258,56.580,413.181,169.624,38.248,157.194
C06665=1040.265,56.830,413.163,169.626,38.249,157.194
C06666=1040.271,57.079,413.145,169.628,38.249,157.195
C06667=1040.277,57.328,413.128,169.630,38.250,157.195
C06668=1040.284,57.577,413.111,169.632,38.251,157.195
C06669=1040.290,57.827,413.093,169.635,38.252,157.195
C06670=1040.296,58.076,413.076,169.636,38.252,157.195
C06671=1040.302,58.326,413.058,169.638,38.253,157.195
C06672=1040.309,58.574,413.041,169.640,38.253,157.196
C06673=1040.316,58.824,413.024,169.642,38.254,157.196
C06674=1040.322,59.074,413.006,169.644,38.254,157.196
C06675=1040.329,59.323,412.989,169.646,38.255,157.196
C06676=1040.334,59.572,412.971,169.647,38.256,157.196
C06677=1040.341,59.822,412.954,169.650,38.257,157.196
C06678=1040.348,60.071,412.936,169.652,38.257,157.196
C06679=1040.353,60.320,412.919,169.654,38.258,157.197
C06680=1040.361,60.607,412.898,169.656,38.258,157.197
C06681=1040.368,60.893,412.878,169.658,38.259,157.197
C06682=1040.375,61.179,412.858,169.660,38.260,157.197
C06683=1040.384,61.466,412.838,169.662,38.261,157.197
C06684=1040.389,61.715,412.821,169.665,38.261,157.197
C06685=1040.396,61.964,412.804,169.667,38.262,157.198
C06686=1040.402,62.213,412.785,169.669,38.262,157.198
C06687=1040.409,62.462,412.768,169.671,38.263,157.198
C06688=1040.415,62.712,412.750,169.673,38.263,157.198
C06689=1040.422,62.961,412.733,169.675,38.264,157.198
C06690=1040.429,63.210,412.715,169.676,38.264,157.198
C06691=1040.435,63.460,412.697,169.678,38.265,157.198
C06692=1040.441,63.709,412.680,169.681,38.266,157.199
C06693=1040.447,63.958,412.662,169.683,38.267,157.199
C06694=1040.454,64.207,412.644,169.685,38.267,157.199
C06695=1040.460,64.457,412.626,169.687,38.268,157.199
C06696=1040.466,64.706,412.609,169.688,38.268,157.199
C06697=1040.473,64.955,412.591,169.690,38.270,157.200
C06698=1040.479,65.205,412.573,169.692,38.270,157.200
C06699=1040.485,65.454,412.555,169.694,38.271,157.200
C06700=1040.492,65.703,412.538,169.697,38.271,157.200
C06701=1040.498,65.952,412.519,169.698,38.272,157.200
C06702=1040.504,66.202,412.501,169.700,38.273,157.200
C06703=1040.510,66.451,412.484,169.702,38.274,157.201
C06704=1040.517,66.700,412.466,169.704,38.274,157.201
C06705=1040.523,66.950,412.448,169.706,38.275,157.201
C06706=1040.529,67.199,412.430,169.708,38.276,157.201
C06707=1040.536,67.448,412.412,169.710,38.276,157.201
C06708=1040.542,67.697,412.394,169.712,38.277,157.201
C06709=1040.548,67.947,412.376,169.714,38.277,157.202
C06710=1040.554,68.196,412.358,169.716,38.279,157.202
C06711=1040.561,68.446,412.340,169.718,38.279,157.202
C06712=1040.567,68.694,412.322,169.719,38.280,157.202
C06713=1040.573,68.944,412.304,169.721,38.280,157.202
C06714=1040.579,69.194,412.286,169.724,38.281,157.202
C06715=1040.586,69.442,412.268,169.726,38.282,157.203
C06716=1040.592,69.692,412.250,169.728,38.283,157.203
C06717=1040.598,69.940,412.232,169.729,38.283,157.203
C06718=1040.604,70.190,412.214,169.731,38.284,157.203
C06719=1040.611,70.439,412.195,169.733,38.285,157.203
C06720=1040.617,70.689,412.177,169.735,38.285,157.203
C06721=1040.623,70.939,412.160,169.738,38.286,157.204
C06722=1040.630,71.187,412.142,169.739,38.287,157.204
C06723=1040.636,71.437,412.124,169.741,38.288,157.204
C06724=1040.642,71.686,412.105,169.743,38.288,157.204
C06725=1040.648,71.936,412.087,169.745,38.289,157.204
C06726=1040.655,72.185,412.069,169.747,38.290,157.205
C06727=1040.661,72.433,412.050,169.748,38.291,157.205
C06728=1040.667,72.683,412.032,169.751,38.291,157.205
C06729=1040.673,72.932,412.014,169.753,38.292,157.205
C06730=1040.679,73.182,411.996,169.755,38.293,157.205
C06731=1040.686,73.431,411.977,169.757,38.293,157.205
C06732=1040.692,73.680,411.960,169.759,38.294,157.206
C06733=1040.698,73.929,411.942,169.760,38.295,157.206
C06734=1040.704,74.178,411.924,169.762,38.296,157.206
C06735=1040.711,74.428,411.905,169.765,38.296,157.206
C06736=1040.717,74.677,411.886,169.767,38.297,157.206
C06737=1040.723,74.926,411.868,169.769,38.298,157.207
C06738=1040.730,75.176,411.850,169.770,38.299,157.207
C06739=1040.736,75.425,411.832,169.772,38.299,157.207
C06740=1040.742,75.674,411.814,169.774,38.300,157.207
C06741=1040.748,75.923,411.795,169.776,38.301,157.207
C06742=1040.754,76.173,411.777,169.779,38.301,157.207
C06743=1040.761,76.422,411.758,169.780,38.302,157.207
C06744=1040.769,76.708,411.737,169.783,38.303,157.208
C06745=1040.775,76.993,411.716,169.785,38.304,157.208
C06746=1040.783,77.280,411.696,169.787,38.305,157.208
C06747=1040.790,77.566,411.674,169.789,38.305,157.208
C06748=1040.796,77.815,411.655,169.792,38.306,157.208
C06749=1040.803,78.064,411.637,169.793,38.307,157.209
C06750=1040.809,78.314,411.619,169.795,38.308,157.209
C06751=1040.815,78.563,411.601,169.797,38.308,157.209
C06752=1040.821,78.812,411.582,169.799,38.309,157.209
C06753=1040.827,79.061,411.563,169.800,38.310,157.209
C06754=1040.833,79.311,411.545,169.803,38.311,157.210
C06755=1040.839,79.560,411.526,169.805,38.312,157.210
C06756=1040.846,79.809,411.507,169.807,38.312,157.210
C06757=1040.852,80.058,411.489,169.809,38.313,157.210
C06758=1040.859,80.307,411.470,169.810,38.314,157.210
C06759=1040.865,80.557,411.452,169.812,38.314,157.211
C06760=1040.870,80.806,411.433,169.814,38.316,157.211
C06761=1040.876,81.055,411.415,169.817,38.316,157.211
C06762=1040.883,81.304,411.396,169.819,38.317,157.211
C06763=1040.889,81.553,411.377,169.820,38.318,157.211
C06764=1040.895,81.802,411.359,169.822,38.318,157.211
C06765=1040.901,82.052,411.340,169.824,38.319,157.212
C06766=1040.907,82.302,411.322,169.826,38.320,157.212
C06767=1040.914,82.551,411.303,169.828,38.321,157.212
C06768=1040.920,82.800,411.284,169.830,38.322,157.212
C06769=1040.927,83.049,411.266,169.832,38.322,157.212
C06770=1040.932,83.298,411.246,169.834,38.323,157.213
C06771=1040.939,83.547,411.228,169.836,38.324,157.213
C06772=1040.945,83.797,411.209,169.838,38.325,157.213
C06773=1040.952,84.046,411.190,169.839,38.325,157.213
C06774=1040.958,84.295,411.172,169.842,38.327,157.213
C06775=1040.963,84.545,411.153,169.844,38.327,157.214
C06776=1040.970,84.794,411.135,169.846,38.328,157.214
C06777=1040.976,85.043,411.116,169.848,38.329,157.214
C06778=1040.983,85.292,411.097,169.849,38.329,157.214
C06779=1040.989,85.541,411.079,169.851,38.330,157.214
C06780=1040.995,85.791,411.059,169.854,38.331,157.215
C06781=1041.001,86.040,411.041,169.856,38.332,157.215
C06782=1041.008,86.289,411.022,169.858,38.332,157.215
C06783=1041.014,86.538,411.003,169.859,38.333,157.215
C06784=1041.020,86.788,410.984,169.861,38.334,157.215
C06785=1041.026,87.037,410.966,169.863,38.334,157.215
C06786=1041.033,87.286,410.947,169.865,38.335,157.215
C06787=1041.039,87.535,410.928,169.868,38.336,157.216
C06788=1041.045,87.769,410.910,169.869,38.337,157.216
C06789=1041.051,88.004,410.892,169.871,38.337,157.216
C06790=1041.057,88.239,410.875,169.873,38.338,157.216
C06791=1041.063,88.473,410.858,169.875,38.339,157.216
C06792=1041.069,88.709,410.839,169.876,38.340,157.217
C06793=1041.075,88.943,410.821,169.878,38.340,157.217
C06794=1041.081,89.178,410.804,169.881,38.341,157.217
C06795=1041.087,89.413,410.786,169.882,38.342,157.217
C06796=1041.092,89.662,410.767,169.884,38.342,157.217
C06797=1041.099,89.911,410.748,169.886,38.343,157.217
C06798=1041.105,90.160,410.729,169.888,38.343,157.218
C06799=1041.111,90.409,410.710,169.890,38.345,157.218
C06800=1041.118,90.658,410.691,169.892,38.345,157.218
C06801=1041.123,90.908,410.672,169.894,38.346,157.218
C06802=1041.130,91.157,410.653,169.896,38.347,157.218
C06803=1041.136,91.406,410.633,169.898,38.348,157.219
C06804=1041.143,91.655,410.614,169.900,38.349,157.219
C06805=1041.148,91.905,410.595,169.901,38.350,157.219
C06806=1041.155,92.154,410.577,169.903,38.350,157.219
C06807=1041.161,92.403,410.557,169.906,38.351,157.219
C06808=1041.169,92.719,410.533,169.908,38.352,157.220
C06809=1041.176,93.032,410.509,169.911,38.353,157.220
C06810=1041.184,93.348,410.484,169.913,38.354,157.220
C06811=1041.192,93.663,410.460,169.915,38.356,157.220
C06812=1041.198,93.912,410.441,169.918,38.356,157.221
C06813=1041.204,94.161,410.422,169.920,38.357,157.221
C06814=1041.210,94.411,410.403,169.922,38.358,157.221
C06815=1041.217,94.659,410.384,169.923,38.358,157.221
C06816=1041.223,94.909,410.364,169.925,38.360,157.221
C06817=1041.229,95.159,410.345,169.927,38.360,157.222
C06818=1041.235,95.407,410.325,169.930,38.361,157.222
C06819=1041.242,95.657,410.307,169.932,38.362,157.222
C06820=1041.248,95.906,410.288,169.933,38.362,157.222
C06821=1041.254,96.154,410.268,169.935,38.364,157.222
C06822=1041.260,96.404,410.249,169.937,38.364,157.223
C06823=1041.267,96.654,410.230,169.939,38.365,157.223
C06824=1041.273,96.903,410.210,169.942,38.366,157.223
C06825=1041.279,97.152,410.191,169.944,38.366,157.223
C06826=1041.285,97.400,410.171,169.945,38.367,157.223
C06827=1041.291,97.650,410.152,169.947,38.368,157.224
C06828=1041.298,97.899,410.133,169.949,38.369,157.224
C06829=1041.304,98.149,410.113,169.951,38.370,157.224
C06830=1041.311,98.398,410.094,169.953,38.370,157.224
C06831=1041.317,98.646,410.074,169.956,38.371,157.224
C06832=1041.323,98.896,410.056,169.957,38.372,157.224
C06833=1041.329,99.145,410.037,169.959,38.373,157.225
C06834=1041.336,99.394,410.017,169.961,38.374,157.225
C06835=1041.342,99.644,409.998,169.963,38.374,157.225
C06836=1041.348,99.892,409.978,169.966,38.375,157.225
C06837=1041.354,100.142,409.959,169.967,38.376,157.225
C06838=1041.360,100.390,409.939,169.969,38.377,157.226
C06839=1041.367,100.640,409.920,169.971,38.378,157.226
C06840=1041.373,100.889,409.900,169.973,38.378,157.226
C06841=1041.379,101.138,409.881,169.975,38.379,157.226
C06842=1041.385,101.387,409.861,169.977,38.380,157.226
C06843=1041.391,101.637,409.842,169.979,38.381,157.227
C06844=1041.398,101.886,409.822,169.981,38.382,157.227
C06845=1041.404,102.135,409.803,169.983,38.383,157.227
C06846=1041.410,102.384,409.783,169.985,38.383,157.227
C06847=1041.416,102.633,409.763,169.987,38.385,157.228
C06848=1041.421,102.882,409.744,169.988,38.385,157.228
C06849=1041.428,103.132,409.723,169.991,38.386,157.228
C06850=1041.434,103.381,409.705,169.993,38.387,157.228
C06851=1041.440,103.630,409.685,169.995,38.388,157.228
C06852=1041.446,103.879,409.665,169.997,38.389,157.228
C06853=1041.452,104.128,409.645,169.998,38.390,157.229
C06854=1041.459,104.378,409.625,170.001,38.390,157.229
C06855=1041.465,104.626,409.606,170.003,38.391,157.229
C06856=1041.471,104.876,409.586,170.005,38.392,157.229
C06857=1041.477,105.124,409.566,170.007,38.393,157.230
C06858=1041.484,105.374,409.546,170.009,38.394,157.230
C06859=1041.489,105.623,409.527,170.010,38.395,157.230
C06860=1041.495,105.872,409.507,170.013,38.395,157.230
C06861=1041.503,106.121,409.487,170.015,38.397,157.230
C06862=1041.508,106.371,409.468,170.017,38.397,157.231
C06863=1041.514,106.620,409.448,170.019,38.398,157.231
C06864=1041.520,106.868,409.428,170.021,38.399,157.231
C06865=1041.527,107.118,409.408,170.022,38.400,157.231
C06866=1041.532,107.367,409.388,170.025,38.401,157.231
C06867=1041.539,107.616,409.369,170.027,38.401,157.232
C06868=1041.546,107.865,409.349,170.029,38.402,157.232
C06869=1041.552,108.114,409.329,170.031,38.403,157.232
C06870=1041.558,108.364,409.310,170.033,38.404,157.232
C06871=1041.564,108.613,409.289,170.034,38.404,157.232
C06872=1041.572,108.899,409.267,170.038,38.406,157.233
C06873=1041.578,109.185,409.244,170.040,38.407,157.233
C06874=1041.586,109.471,409.222,170.042,38.407,157.233
C06875=1041.592,109.757,409.199,170.044,38.408,157.233
C06876=1041.599,110.006,409.178,170.046,38.409,157.233
C06877=1041.605,110.255,409.158,170.049,38.410,157.234
C06878=1041.611,110.504,409.138,170.051,38.411,157.234
C06879=1041.618,110.753,409.119,170.052,38.412,157.234
C06880=1041.624,111.002,409.099,170.054,38.412,157.234
C06881=1041.630,111.251,409.080,170.056,38.414,157.235
C06882=1041.637,111.501,409.059,170.058,38.414,157.235
C06883=1041.643,111.749,409.039,170.061,38.415,157.235
C06884=1041.649,111.999,409.019,170.063,38.416,157.235
C06885=1041.655,112.248,408.999,170.064,38.417,157.235
C06886=1041.661,112.497,408.979,170.066,38.418,157.236
C06887=1041.668,112.746,408.959,170.068,38.419,157.236
C06888=1041.673,112.995,408.938,170.071,38.420,157.236
C06889=1041.679,113.244,408.918,170.073,38.420,157.236
C06890=1041.686,113.494,408.898,170.075,38.422,157.237
C06891=1041.692,113.742,408.878,170.077,38.422,157.237
C06892=1041.698,113.991,408.858,170.078,38.423,157.237
C06893=1041.704,114.241,408.838,170.080,38.424,157.237
C06894=1041.709,114.490,408.817,170.083,38.425,157.237
C06895=1041.715,114.739,408.797,170.085,38.426,157.238
C06896=1041.722,114.988,408.777,170.087,38.427,157.238
C06897=1041.728,115.237,408.757,170.088,38.428,157.238
C06898=1041.733,115.486,408.736,170.090,38.429,157.238
C06899=1041.740,115.736,408.716,170.093,38.430,157.239
C06900=1041.746,115.984,408.696,170.095,38.431,157.239
C06901=1041.752,116.234,408.676,170.097,38.432,157.239
C06902=1041.758,116.483,408.655,170.099,38.432,157.239
C06903=1041.764,116.732,408.635,170.100,38.434,157.239
C06904=1041.771,116.981,408.614,170.103,38.435,157.240
C06905=1041.776,117.230,408.594,170.105,38.435,157.240
C06906=1041.782,117.479,408.573,170.107,38.436,157.240
C06907=1041.788,117.728,408.553,170.109,38.438,157.240
C06908=1041.794,117.977,408.533,170.111,38.438,157.241
C06909=1041.800,118.227,408.512,170.114,38.439,157.241
C06910=1041.806,118.476,408.492,170.115,38.440,157.241
C06911=1041.813,118.725,408.471,170.117,38.441,157.241
C06912=1041.818,118.974,408.451,170.119,38.442,157.241
C06913=1041.824,119.223,408.431,170.121,38.443,157.242
C06914=1041.831,119.472,408.411,170.123,38.444,157.242
C06915=1041.837,119.721,408.391,170.126,38.445,157.242
C06916=1041.843,119.970,408.369,170.128,38.446,157.242
C06917=1041.849,120.219,408.349,170.129,38.447,157.243
C06918=1041.856,120.468,408.329,170.131,38.448,157.243
C06919=1041.861,120.717,408.308,170.133,38.448,157.243
C06920=1041.868,120.966,408.287,170.136,38.450,157.243
C06921=1041.874,121.215,408.267,170.138,38.450,157.243
C06922=1041.880,121.465,408.246,170.140,38.451,157.244
C06923=1041.886,121.714,408.226,170.142,38.452,157.244
C06924=1041.893,121.963,408.205,170.143,38.453,157.244
C06925=1041.899,122.212,408.185,170.146,38.454,157.244
C06926=1041.904,122.461,408.165,170.148,38.455,157.245
C06927=1041.911,122.710,408.144,170.150,38.456,157.245
C06928=1041.917,122.959,408.123,170.152,38.457,157.245
C06929=1041.923,123.208,408.103,170.154,38.458,157.245
C06930=1041.929,123.458,408.082,170.156,38.459,157.245
C06931=1041.936,123.706,408.062,170.159,38.460,157.246
C06932=1041.941,123.956,408.041,170.161,38.460,157.246
C06933=1041.947,124.205,408.021,170.162,38.462,157.246
C06934=1041.954,124.453,408.000,170.164,38.462,157.246
C06935=1041.960,124.703,407.979,170.166,38.463,157.247
C06936=1041.967,124.989,407.955,170.169,38.464,157.247
C06937=1041.974,125.274,407.932,170.172,38.465,157.247
C06938=1041.981,125.560,407.909,170.174,38.466,157.247
C06939=1041.989,125.846,407.885,170.176,38.467,157.248
C06940=1041.995,126.094,407.864,170.178,38.468,157.248
C06941=1042.001,126.344,407.843,170.181,38.469,157.248
C06942=1042.007,126.594,407.823,170.183,38.470,157.248
C06943=1042.014,126.842,407.802,170.185,38.471,157.249
C06944=1042.019,127.092,407.781,170.186,38.472,157.249
C06945=1042.026,127.340,407.760,170.188,38.473,157.249
C06946=1042.032,127.589,407.740,170.191,38.473,157.249
C06947=1042.038,127.839,407.718,170.193,38.475,157.249
C06948=1042.044,128.087,407.699,170.195,38.476,157.250
C06949=1042.051,128.337,407.677,170.197,38.476,157.250
C06950=1042.057,128.585,407.657,170.199,38.477,157.250
C06951=1042.064,128.834,407.636,170.201,38.478,157.250
C06952=1042.069,129.084,407.615,170.204,38.479,157.250
C06953=1042.076,129.332,407.594,170.206,38.480,157.251
C06954=1042.082,129.582,407.574,170.208,38.481,157.251
C06955=1042.088,129.831,407.552,170.210,38.482,157.251
C06956=1042.094,130.080,407.532,170.212,38.482,157.251
C06957=1042.101,130.329,407.511,170.214,38.484,157.252
C06958=1042.107,130.579,407.490,170.216,38.484,157.252
C06959=1042.113,130.827,407.470,170.218,38.485,157.252
C06960=1042.120,131.076,407.449,170.220,38.486,157.252
C06961=1042.126,131.326,407.428,170.222,38.487,157.252
C06962=1042.132,131.574,407.407,170.225,38.488,157.253
C06963=1042.138,131.824,407.386,170.227,38.489,157.253
C06964=1042.144,132.072,407.365,170.229,38.490,157.253
C06965=1042.150,132.321,407.343,170.231,38.491,157.253
C06966=1042.157,132.571,407.323,170.233,38.492,157.254
C06967=1042.162,132.819,407.302,170.236,38.493,157.254
C06968=1042.168,133.069,407.280,170.238,38.494,157.254
C06969=1042.175,133.318,407.260,170.240,38.495,157.254
C06970=1042.181,133.567,407.238,170.241,38.496,157.255
C06971=1042.187,133.816,407.217,170.243,38.497,157.255
C06972=1042.194,134.065,407.196,170.246,38.498,157.255
C06973=1042.199,134.314,407.175,170.248,38.499,157.255
C06974=1042.205,134.563,407.154,170.250,38.500,157.256
C06975=1042.212,134.812,407.133,170.252,38.501,157.256
C06976=1042.218,135.060,407.111,170.254,38.502,157.256
C06977=1042.223,135.310,407.090,170.257,38.503,157.256
C06978=1042.230,135.559,407.069,170.259,38.504,157.257
C06979=1042.236,135.808,407.048,170.261,38.505,157.257
C06980=1042.242,136.057,407.026,170.263,38.506,157.257
C06981=1042.248,136.307,407.006,170.266,38.507,157.257
C06982=1042.254,136.555,406.985,170.268,38.508,157.258
C06983=1042.260,136.804,406.963,170.270,38.509,157.258
C06984=1042.267,137.053,406.942,170.272,38.510,157.258
C06985=1042.273,137.302,406.921,170.273,38.511,157.258
C06986=1042.279,137.551,406.899,170.276,38.512,157.259
C06987=1042.285,137.800,406.878,170.278,38.513,157.259
C06988=1042.291,138.050,406.857,170.280,38.514,157.259
C06989=1042.297,138.298,406.836,170.282,38.515,157.259
C06990=1042.303,138.547,406.814,170.284,38.516,157.260
C06991=1042.310,138.796,406.793,170.287,38.517,157.260
C06992=1042.316,139.045,406.771,170.289,38.518,157.260
C06993=1042.322,139.294,406.750,170.291,38.519,157.260
C06994=1042.328,139.543,406.729,170.293,38.520,157.260
C06995=1042.334,139.792,406.707,170.295,38.521,157.261
C06996=1042.341,140.041,406.686,170.298,38.522,157.261
C06997=1042.346,140.290,406.664,170.300,38.523,157.261
C06998=1042.352,140.539,406.643,170.302,38.524,157.261
C06999=1042.358,140.788,406.621,170.304,38.525,157.262
C07000=1042.365,141.074,406.597,170.307,38.526,157.262
C07001=1042.373,141.359,406.572,170.309,38.527,157.262
C07002=1042.379,141.645,406.548,170.312,38.528,157.263
C07003=1042.386,141.931,406.522,170.314,38.530,157.263
C07004=1042.392,142.180,406.501,170.316,38.531,157.263
C07005=1042.398,142.429,406.479,170.319,38.532,157.263
C07006=1042.404,142.678,406.458,170.321,38.533,157.264
C07007=1042.411,142.927,406.437,170.323,38.534,157.264
C07008=1042.417,143.176,406.415,170.325,38.535,157.264
C07009=1042.423,143.425,406.394,170.328,38.536,157.264
C07010=1042.430,143.674,406.371,170.330,38.537,157.265
C07011=1042.435,143.922,406.350,170.332,38.538,157.265
C07012=1042.441,144.171,406.328,170.334,38.539,157.265
C07013=1042.448,144.421,406.307,170.336,38.540,157.265
C07014=1042.454,144.670,406.285,170.339,38.541,157.266
C07015=1042.460,144.919,406.263,170.340,38.542,157.266
C07016=1042.465,145.168,406.242,170.342,38.543,157.266
C07017=1042.472,145.417,406.221,170.344,38.544,157.266
C07018=1042.478,145.665,406.198,170.347,38.546,157.267
C07019=1042.484,145.915,406.177,170.349,38.547,157.267
C07020=1042.490,146.164,406.155,170.351,38.547,157.267
C07021=1042.497,146.413,406.133,170.353,38.548,157.267
C07022=1042.503,146.662,406.112,170.355,38.549,157.268
C07023=1042.509,146.910,406.090,170.358,38.551,157.268
C07024=1042.515,147.159,406.068,170.360,38.552,157.268
C07025=1042.521,147.408,406.046,170.362,38.553,157.269
C07026=1042.527,147.658,406.025,170.364,38.554,157.269
C07027=1042.534,147.906,406.002,170.366,38.555,157.269
C07028=1042.540,148.155,405.981,170.369,38.556,157.269
C07029=1042.546,148.405,405.959,170.371,38.557,157.270
C07030=1042.552,148.654,405.937,170.373,38.558,157.270
C07031=1042.557,148.902,405.915,170.375,38.559,157.270
C07032=1042.563,149.151,405.893,170.378,38.560,157.270
C07033=1042.570,149.400,405.872,170.380,38.561,157.271
C07034=1042.576,149.649,405.849,170.382,38.563,157.271
C07035=1042.582,149.898,405.828,170.384,38.564,157.271
C07036=1042.589,150.147,405.805,170.388,38.565,157.271
C07037=1042.594,150.396,405.783,170.390,38.566,157.272
C07038=1042.600,150.646,405.761,170.392,38.567,157.272
C07039=1042.607,150.894,405.739,170.394,38.568,157.272
C07040=1042.612,151.143,405.718,170.397,38.569,157.273
C07041=1042.619,151.391,405.695,170.399,38.570,157.273
C07042=1042.624,151.641,405.673,170.401,38.571,157.273
C07043=1042.630,151.890,405.652,170.403,38.572,157.273
C07044=1042.637,152.139,405.629,170.405,38.573,157.274
C07045=1042.643,152.388,405.608,170.408,38.574,157.274
C07046=1042.649,152.636,405.585,170.410,38.576,157.274
C07047=1042.655,152.886,405.563,170.412,38.577,157.274
C07048=1042.661,153.134,405.541,170.414,38.578,157.275
C07049=1042.667,153.384,405.519,170.417,38.579,157.275
C07050=1042.674,153.632,405.497,170.419,38.580,157.275
C07051=1042.679,153.882,405.474,170.421,38.581,157.275
C07052=1042.686,154.130,405.452,170.423,38.582,157.276
C07053=1042.692,154.380,405.430,170.426,38.584,157.276
C07054=1042.698,154.628,405.408,170.428,38.585,157.276
C07055=1042.704,154.878,405.386,170.430,38.586,157.277
C07056=1042.710,155.126,405.364,170.432,38.587,157.277
C07057=1042.716,155.375,405.342,170.435,38.588,157.277
C07058=1042.722,155.624,405.319,170.437,38.589,157.277
C07059=1042.729,155.873,405.297,170.439,38.590,157.278
C07060=1042.734,156.122,405.274,170.441,38.592,157.278
C07061=1042.741,156.371,405.252,170.443,38.593,157.278
C07062=1042.747,156.620,405.230,170.446,38.594,157.279
C07063=1042.752,156.869,405.207,170.448,38.595,157.279
C07064=1042.759,157.154,405.182,170.451,38.596,157.279
C07065=1042.767,157.439,405.156,170.454,38.598,157.280
C07066=1042.774,157.725,405.131,170.457,38.599,157.280
C07067=1042.781,158.010,405.105,170.459,38.600,157.280
C07068=1042.786,158.258,405.082,170.461,38.601,157.280
C07069=1042.792,158.508,405.061,170.464,38.602,157.281
C07070=1042.799,158.756,405.038,170.466,38.603,157.281
C07071=1042.805,159.005,405.016,170.468,38.605,157.281
C07072=1042.811,159.254,404.994,170.470,38.606,157.281
C07073=1042.817,159.503,404.971,170.472,38.607,157.282
C07074=1042.824,159.753,404.948,170.475,38.608,157.282
C07075=1042.830,160.001,404.926,170.478,38.609,157.282
C07076=1042.836,160.251,404.904,170.480,38.610,157.283
C07077=1042.842,160.499,404.881,170.483,38.612,157.283
C07078=1042.848,160.748,404.858,170.485,38.613,157.283
C07079=1042.853,160.997,404.835,170.487,38.614,157.284
C07080=1042.859,161.246,404.812,170.489,38.615,157.284
C07081=1042.865,161.495,404.790,170.492,38.617,157.284
C07082=1042.871,161.743,404.767,170.494,38.618,157.285
C07083=1042.877,161.993,404.745,170.496,38.619,157.285
C07084=1042.883,162.242,404.722,170.498,38.620,157.285
C07085=1042.888,162.491,404.699,170.501,38.622,157.285
C07086=1042.895,162.739,404.677,170.503,38.623,157.286
C07087=1042.901,162.988,404.654,170.505,38.624,157.286
C07088=1042.906,163.237,404.631,170.507,38.626,157.286
C07089=1042.912,163.486,404.608,170.510,38.627,157.287
C07090=1042.918,163.735,404.585,170.512,38.629,157.287
C07091=1042.924,163.983,404.563,170.514,38.630,157.287
C07092=1042.930,164.232,404.540,170.518,38.631,157.288
C07093=1042.936,164.481,404.517,170.520,38.632,157.288
C07094=1042.941,164.730,404.494,170.522,38.634,157.288
C07095=1042.947,164.979,404.471,170.524,38.635,157.289
C07096=1042.954,165.228,404.448,170.527,38.636,157.289
C07097=1042.960,165.477,404.425,170.529,38.638,157.289
C07098=1042.966,165.726,404.402,170.531,38.639,157.290
C07099=1042.971,165.975,404.379,170.533,38.640,157.290
C07100=1042.977,166.224,404.356,170.536,38.641,157.290
C07101=1042.984,166.473,404.334,170.538,38.643,157.290
C07102=1042.990,166.721,404.310,170.540,38.644,157.291
C07103=1042.995,166.970,404.287,170.544,38.645,157.291
C07104=1043.001,167.219,404.264,170.546,38.646,157.291
C07105=1043.007,167.468,404.241,170.548,38.648,157.292
C07106=1043.014,167.717,404.219,170.550,38.649,157.292
C07107=1043.020,167.966,404.196,170.553,38.650,157.292
C07108=1043.025,168.215,404.173,170.555,38.651,157.293
C07109=1043.031,168.463,404.150,170.557,38.653,157.293
C07110=1043.037,168.712,404.126,170.559,38.654,157.293
C07111=1043.043,168.961,404.103,170.563,38.655,157.294
C07112=1043.050,169.210,404.081,170.565,38.656,157.294
C07113=1043.056,169.459,404.058,170.567,38.658,157.294
C07114=1043.061,169.708,404.035,170.570,38.659,157.295
C07115=1043.067,169.956,404.011,170.572,38.660,157.295
C07116=1043.074,170.206,403.988,170.574,38.662,157.295
C07117=1043.079,170.455,403.965,170.576,38.663,157.295
C07118=1043.086,170.703,403.942,170.580,38.664,157.296
C07119=1043.092,170.952,403.919,170.582,38.665,157.296
C07120=1043.098,171.200,403.896,170.584,38.667,157.296
C07121=1043.104,171.450,403.872,170.587,38.668,157.297
C07122=1043.110,171.699,403.850,170.589,38.669,157.297
C07123=1043.116,171.947,403.826,170.591,38.671,157.297
C07124=1043.122,172.196,403.803,170.594,38.672,157.298
C07125=1043.129,172.445,403.780,170.597,38.673,157.298
C07126=1043.134,172.694,403.757,170.599,38.675,157.298
C07127=1043.140,172.942,403.734,170.601,38.676,157.299
C07128=1043.147,173.228,403.707,170.604,38.677,157.299
C07129=1043.155,173.512,403.680,170.607,38.679,157.299
C07130=1043.161,173.797,403.654,170.610,38.680,157.300
C07131=1043.169,174.082,403.628,170.612,38.682,157.300
C07132=1043.175,174.331,403.604,170.615,38.683,157.300
C07133=1043.181,174.580,403.581,170.617,38.685,157.301
C07134=1043.187,174.828,403.557,170.620,38.686,157.301
C07135=1043.193,175.077,403.534,170.623,38.687,157.301
C07136=1043.199,175.327,403.511,170.625,38.689,157.302
C07137=1043.205,175.575,403.487,170.627,38.690,157.302
C07138=1043.211,175.824,403.464,170.629,38.691,157.302
C07139=1043.217,176.073,403.440,170.633,38.692,157.303
C07140=1043.224,176.322,403.418,170.635,38.694,157.303
C07141=1043.230,176.570,403.394,170.637,38.695,157.303
C07142=1043.236,176.820,403.371,170.640,38.696,157.304
C07143=1043.242,177.068,403.347,170.643,38.698,157.304
C07144=1043.248,177.317,403.324,170.645,38.699,157.304
C07145=1043.255,177.566,403.300,170.647,38.700,157.305
C07146=1043.260,177.815,403.277,170.650,38.702,157.305
C07147=1043.267,178.064,403.253,170.652,38.703,157.305
C07148=1043.273,178.313,403.230,170.655,38.704,157.306
C07149=1043.280,178.560,403.207,170.658,38.706,157.306
C07150=1043.286,178.810,403.184,170.660,38.707,157.306
C07151=1043.292,179.058,403.160,170.662,38.708,157.307
C07152=1043.298,179.308,403.137,170.665,38.709,157.307
C07153=1043.304,179.556,403.113,170.668,38.711,157.307
C07154=1043.311,179.805,403.089,170.670,38.712,157.307
C07155=1043.317,180.054,403.066,170.672,38.713,157.308
C07156=1043.323,180.302,403.043,170.676,38.715,157.308
C07157=1043.329,180.552,403.019,170.678,38.716,157.308
C07158=1043.335,180.800,402.996,170.680,38.717,157.309
C07159=1043.342,181.049,402.972,170.683,38.719,157.309
C07160=1043.347,181.298,402.949,170.686,38.720,157.309
C07161=1043.355,181.547,402.925,170.688,38.721,157.310
C07162=1043.361,181.795,402.902,170.690,38.723,157.310
C07163=1043.367,182.045,402.878,170.694,38.724,157.310
C07164=1043.373,182.293,402.855,170.696,38.725,157.311
C07165=1043.380,182.542,402.831,170.698,38.726,157.311
C07166=1043.386,182.791,402.808,170.701,38.728,157.311
C07167=1043.392,183.040,402.784,170.704,38.729,157.312
C07168=1043.398,183.288,402.760,170.706,38.730,157.312
C07169=1043.405,183.538,402.737,170.708,38.732,157.312
C07170=1043.411,183.786,402.713,170.712,38.733,157.313
C07171=1043.416,184.035,402.689,170.714,38.734,157.313
C07172=1043.423,184.284,402.665,170.716,38.736,157.314
C07173=1043.429,184.532,402.641,170.719,38.738,157.314
C07174=1043.434,184.781,402.617,170.722,38.739,157.314
C07175=1043.441,185.030,402.593,170.724,38.741,157.315
C07176=1043.446,185.279,402.568,170.727,38.742,157.315
C07177=1043.452,185.527,402.545,170.729,38.743,157.315
C07178=1043.458,185.776,402.520,170.732,38.745,157.316
C07179=1043.464,186.024,402.496,170.735,38.747,157.316
C07180=1043.470,186.274,402.472,170.737,38.748,157.316
C07181=1043.476,186.523,402.449,170.739,38.750,157.317
C07182=1043.482,186.772,402.424,170.743,38.751,157.317
C07183=1043.488,187.020,402.401,170.745,38.753,157.318
C07184=1043.494,187.269,402.375,170.747,38.754,157.318
C07185=1043.500,187.517,402.352,170.751,38.756,157.318
C07186=1043.506,187.766,402.327,170.753,38.757,157.319
C07187=1043.512,188.015,402.303,170.755,38.759,157.319
C07188=1043.518,188.264,402.279,170.758,38.761,157.320
C07189=1043.524,188.512,402.255,170.761,38.762,157.320
C07190=1043.530,188.762,402.230,170.763,38.763,157.320
C07191=1043.536,189.010,402.207,170.766,38.765,157.321
C07192=1043.543,189.295,402.179,170.769,38.767,157.321
C07193=1043.550,189.579,402.151,170.772,38.768,157.321
C07194=1043.557,189.864,402.123,170.775,38.770,157.322
C07195=1043.563,190.148,402.096,170.778,38.772,157.322
C07196=1043.569,190.397,402.071,170.780,38.774,157.323
C07197=1043.575,190.645,402.047,170.784,38.775,157.323
C07198=1043.581,190.894,402.023,170.786,38.776,157.323
C07199=1043.588,191.143,401.999,170.788,38.778,157.324
C07200=1043.594,191.391,401.974,170.791,38.780,157.324
C07201=1043.600,191.640,401.950,170.794,38.781,157.325
C07202=1043.605,191.889,401.925,170.796,38.783,157.325
C07203=1043.612,192.138,401.901,170.799,38.784,157.325
C07204=1043.618,192.387,401.877,170.802,38.786,157.326
C07205=1043.624,192.635,401.852,170.804,38.788,157.326
C07206=1043.630,192.884,401.828,170.808,38.789,157.327
C07207=1043.636,193.132,401.804,170.810,38.791,157.327
C07208=1043.643,193.381,401.779,170.812,38.792,157.327
C07209=1043.649,193.630,401.755,170.816,38.794,157.328
C07210=1043.654,193.879,401.730,170.818,38.795,157.328
C07211=1043.660,194.128,401.706,170.820,38.797,157.328
C07212=1043.667,194.376,401.681,170.824,38.798,157.329
C07213=1043.673,194.625,401.657,170.826,38.800,157.329
C07214=1043.679,194.874,401.633,170.828,38.801,157.330
C07215=1043.685,195.123,401.607,170.832,38.803,157.330
C07216=1043.692,195.372,401.583,170.834,38.805,157.330
C07217=1043.697,195.620,401.559,170.838,38.806,157.331
C07218=1043.704,195.869,401.534,170.840,38.807,157.331
C07219=1043.710,196.118,401.510,170.842,38.809,157.332
C07220=1043.716,196.366,401.485,170.846,38.811,157.332
C07221=1043.722,196.615,401.461,170.848,38.813,157.332
C07222=1043.728,196.864,401.436,170.851,38.814,157.333
C07223=1043.735,197.112,401.411,170.854,38.815,157.333
C07224=1043.741,197.361,401.387,170.856,38.817,157.334
C07225=1043.748,197.609,401.362,170.859,38.819,157.334
C07226=1043.753,197.859,401.338,170.862,38.821,157.334
C07227=1043.760,198.107,401.312,170.865,38.822,157.335
C07228=1043.766,198.356,401.289,170.867,38.823,157.335
C07229=1043.772,198.604,401.263,170.870,38.825,157.335
C07230=1043.779,198.853,401.239,170.873,38.827,157.336
C07231=1043.785,199.102,401.214,170.875,38.828,157.336
C07232=1043.791,199.351,401.189,170.879,38.830,157.337
C07233=1043.797,199.599,401.165,170.881,38.832,157.337
C07234=1043.803,199.848,401.140,170.884,38.833,157.337
C07235=1043.810,200.097,401.116,170.887,38.835,157.338
C07236=1043.816,200.346,401.091,170.889,38.836,157.338
C07237=1043.823,200.594,401.066,170.893,38.838,157.339
C07238=1043.829,200.843,401.041,170.895,38.840,157.339
C07239=1043.834,201.091,401.017,170.898,38.841,157.340
C07240=1043.841,201.340,400.992,170.901,38.843,157.340
C07241=1043.847,201.589,400.967,170.904,38.845,157.340
C07242=1043.853,201.838,400.942,170.906,38.846,157.341
C07243=1043.859,202.086,400.917,170.910,38.848,157.341
C07244=1043.866,202.335,400.891,170.912,38.850,157.342
C07245=1043.871,202.584,400.867,170.915,38.852,157.342
C07246=1043.877,202.832,400.842,170.918,38.853,157.342
C07247=1043.883,203.081,400.816,170.920,38.855,157.343
C07248=1043.890,203.330,400.791,170.924,38.857,157.343
C07249=1043.895,203.579,400.767,170.926,38.858,157.344
C07250=1043.902,203.828,400.741,170.929,38.860,157.344
C07251=1043.907,204.076,400.716,170.932,38.862,157.345
C07252=1043.914,204.324,400.691,170.935,38.863,157.345
C07253=1043.920,204.573,400.666,170.938,38.865,157.345
C07254=1043.927,204.821,400.641,170.940,38.867,157.346
C07255=1043.933,205.071,400.616,170.943,38.868,157.346
C07256=1043.959,206.122,400.509,171.208,38.971,157.375
C07257=1043.966,206.407,400.479,171.211,38.973,157.375
C07258=1043.974,206.692,400.449,171.213,38.976,157.376
C07259=1043.982,206.977,400.419,171.216,38.979,157.376
C07260=1043.989,207.263,400.388,171.219,38.982,157.377
C07261=1043.995,207.512,400.363,171.220,38.984,157.378
C07262=1044.003,207.760,400.336,171.223,38.987,157.378
C07263=1044.008,208.009,400.310,171.224,38.989,157.379
C07264=1044.015,208.257,400.283,171.227,38.992,157.379
C07265=1044.022,208.505,400.257,171.229,38.994,157.380
C07266=1044.028,208.755,400.230,171.231,38.997,157.381
C07267=1044.035,209.003,400.204,171.234,38.999,157.381
C07268=1044.042,209.251,400.178,171.235,39.002,157.382
C07269=1044.048,209.500,400.151,171.238,39.004,157.382
C07270=1044.055,209.748,400.125,171.239,39.007,157.383
C07271=1044.061,209.996,400.099,171.242,39.009,157.384
C07272=1044.068,210.245,400.071,171.244,39.012,157.384
C07273=1044.075,210.493,400.045,171.246,39.014,157.385
C07274=1044.082,210.742,400.018,171.248,39.017,157.385
C07275=1044.087,210.990,399.992,171.250,39.019,157.386
C07276=1044.095,211.239,399.965,171.252,39.022,157.386
C07277=1044.101,211.488,399.938,171.255,39.024,157.387
C07278=1044.107,211.736,399.912,171.256,39.027,157.388
C07279=1044.115,211.985,399.886,171.259,39.029,157.388
C07280=1044.120,212.233,399.859,171.262,39.032,157.389
C07281=1044.127,212.481,399.831,171.263,39.035,157.389
C07282=1044.133,212.730,399.805,171.266,39.037,157.390
C07283=1044.140,212.979,399.778,171.267,39.039,157.390
C07284=1044.147,213.227,399.752,171.270,39.042,157.391
C07285=1044.153,213.476,399.725,171.272,39.044,157.392
C07286=1044.160,213.724,399.698,171.274,39.047,157.392
C07287=1044.166,213.972,399.671,171.276,39.049,157.393
C07288=1044.173,214.221,399.645,171.279,39.052,157.393
